LIN {X 0,Y 354.902,Z 376.278,A -85,B 0,C 180,E1 -13615.827,E2 -13615.827} C_VEL
LIN {X 0,Y 354.82,Z 376.288,A -85,B 0,C 180,E1 -13619.682,E2 -13619.682} C_VEL
LIN {X 0,Y 354.808,Z 376.29,A -85,B 0,C 180,E1 -13623.702,E2 -13623.702} C_VEL
LIN {X 0,Y 354.803,Z 376.287,A -85,B 0,C 180,E1 -13626.459,E2 -13626.459} C_VEL
LIN {X 0,Y 354.826,Z 376.289,A -85,B 0,C 180,E1 -13629.423,E2 -13629.423} C_VEL
LIN {X 0,Y 354.79,Z 376.29,A -85,B 0,C 180,E1 -13632.867,E2 -13632.867} C_VEL
LIN {X 0,Y 354.769,Z 376.291,A -85,B 0,C 180,E1 -13636.104,E2 -13636.104} C_VEL
LIN {X 0,Y 354.79,Z 376.293,A -85,B 0,C 180,E1 -13639.179,E2 -13639.179} C_VEL
LIN {X 0,Y 354.809,Z 376.286,A -85,B 0,C 180,E1 -13642.402,E2 -13642.402} C_VEL
LIN {X 0,Y 354.8,Z 376.288,A -85,B 0,C 180,E1 -13643.688,E2 -13643.688} C_VEL
LIN {X 0,Y 354.142,Z 376.373,A -85,B 0,C 180,E1 -13644.636,E2 -13644.636} C_VEL
LIN {X 0,Y 351.287,Z 376.725,A -85,B 0,C 180,E1 -13646.177,E2 -13646.177} C_VEL
LIN {X 0,Y 348.861,Z 377.029,A -85,B 0,C 180,E1 -13647.425,E2 -13647.425} C_VEL
LIN {X 0,Y 347.817,Z 377.158,A -85,B 0,C 180,E1 -13648.39,E2 -13648.39} C_VEL
LIN {X 0,Y 347.732,Z 377.165,A -85,B 0,C 180,E1 -13648.717,E2 -13648.717} C_VEL
LIN {X 0,Y 347.807,Z 377.163,A -85,B 0,C 180,E1 -13650.99,E2 -13650.99} C_VEL
LIN {X 0,Y 347.834,Z 377.155,A -85,B 0,C 180,E1 -13653.608,E2 -13653.608} C_VEL
LIN {X 0,Y 347.791,Z 377.16,A -85,B 0,C 180,E1 -13656.162,E2 -13656.162} C_VEL
LIN {X 0,Y 347.815,Z 377.157,A -85,B 0,C 180,E1 -13659.909,E2 -13659.909} C_VEL
LIN {X 0,Y 347.868,Z 377.152,A -85,B 0,C 180,E1 -13662.359,E2 -13662.359} C_VEL
LIN {X 0,Y 347.899,Z 377.147,A -85,B 0,C 180,E1 -13665.971,E2 -13665.971} C_VEL
LIN {X 0,Y 347.935,Z 377.142,A -85,B 0,C 180,E1 -13669.526,E2 -13669.526} C_VEL
LIN {X 0,Y 348.077,Z 377.125,A -85,B 0,C 180,E1 -13671.875,E2 -13671.875} C_VEL
LIN {X 0,Y 348.07,Z 377.128,A -85,B 0,C 180,E1 -13674.206,E2 -13674.206} C_VEL
LIN {X 0,Y 348.208,Z 377.108,A -85,B 0,C 180,E1 -13677.686,E2 -13677.686} C_VEL
LIN {X 0,Y 348.349,Z 377.092,A -85,B 0,C 180,E1 -13680,E2 -13680} C_VEL
LIN {X 0,Y 348.21,Z 377.112,A -85,B 0,C 180,E1 -13682.313,E2 -13682.313} C_VEL
LIN {X 0,Y 348.108,Z 377.121,A -85,B 0,C 180,E1 -13686.958,E2 -13686.958} C_VEL
LIN {X 0,Y 347.969,Z 377.138,A -85,B 0,C 180,E1 -13689.298,E2 -13689.298} C_VEL
LIN {X 0,Y 347.892,Z 377.149,A -85,B 0,C 180,E1 -13692.839,E2 -13692.839} C_VEL
LIN {X 0,Y 347.841,Z 377.157,A -85,B 0,C 180,E1 -13696.431,E2 -13696.431} C_VEL
LIN {X 0,Y 347.857,Z 377.152,A -85,B 0,C 180,E1 -13698.86,E2 -13698.86} C_VEL
LIN {X 0,Y 347.776,Z 377.164,A -85,B 0,C 180,E1 -13702.579,E2 -13702.579} C_VEL
LIN {X 0,Y 347.814,Z 377.157,A -85,B 0,C 180,E1 -13705.108,E2 -13705.108} C_VEL
LIN {X 0,Y 347.809,Z 377.16,A -85,B 0,C 180,E1 -13707.694,E2 -13707.694} C_VEL
LIN {X 0,Y 347.75,Z 377.168,A -85,B 0,C 180,E1 -13710.348,E2 -13710.348} C_VEL
LIN {X 0,Y 347.749,Z 377.17,A -85,B 0,C 180,E1 -13714.044,E2 -13714.044} C_VEL
LIN {X 0,Y 347.764,Z 377.165,A -85,B 0,C 180,E1 -13717.321,E2 -13717.321} C_VEL
LIN {X 0,Y 347.745,Z 377.167,A -85,B 0,C 180,E1 -13720.295,E2 -13720.295} C_VEL
LIN {X 0,Y 347.726,Z 377.171,A -85,B 0,C 180,E1 -13723.408,E2 -13723.408} C_VEL
LIN {X 0,Y 347.747,Z 377.166,A -85,B 0,C 180,E1 -13726.683,E2 -13726.683} C_VEL
LIN {X 0,Y 347.749,Z 377.166,A -85,B 0,C 180,E1 -13730.173,E2 -13730.173} C_VEL
LIN {X 0,Y 347.822,Z 377.188,A -85,B 0,C 180,E1 -13731.43,E2 -13731.43} C_VEL
LIN {X 0,Y 350.046,Z 388.259,A -85,B 0,C 180,E1 -13735.404,E2 -13735.404} C_VEL
LIN {X 0,Y 352.34,Z 398.991,A -85,B 0,C 180,E1 -13739.06,E2 -13739.06} C_VEL
LIN {X 0,Y 352.6,Z 402.242,A -85,B 0,C 180,E1 -13740.112,E2 -13740.112} C_VEL
LIN {X 0,Y 350.956,Z 413.413,A -85,B 0,C 180,E1 -13743.541,E2 -13743.541} C_VEL
LIN {X 0,Y 349.245,Z 426.523,A -85,B 0,C 180,E1 -13747.521,E2 -13747.521} C_VEL
LIN {X 0,Y 347.88,Z 441.264,A -85,B 0,C 180,E1 -13751.933,E2 -13751.933} C_VEL
LIN {X 0,Y 348.663,Z 454.689,A -85,B 0,C 180,E1 -13752.458,E2 -13752.458} C_VEL
LIN {X 0,Y 349.685,Z 467.492,A -85,B 0,C 180,E1 -13753.207,E2 -13753.207} C_VEL
LIN {X 0,Y 349.831,Z 473.774,A -85,B 0,C 180,E1 -13753.665,E2 -13753.665} C_VEL
LIN {X 0,Y 349.134,Z 485.339,A -85,B 0,C 180,E1 -13754.68,E2 -13754.68} C_VEL
LIN {X 0,Y 348.486,Z 495.132,A -85,B 0,C 180,E1 -13755.772,E2 -13755.772} C_VEL
LIN {X 0,Y 347.817,Z 505.176,A -85,B 0,C 180,E1 -13757.158,E2 -13757.158} C_VEL
LIN {X 0,Y 347.265,Z 513.742,A -85,B 0,C 180,E1 -13758.62,E2 -13758.62} C_VEL
LIN {X 0,Y 346.833,Z 521.96,A -85,B 0,C 180,E1 -13760.377,E2 -13760.377} C_VEL
LIN {X 0,Y 346.716,Z 527.501,A -85,B 0,C 180,E1 -13761.843,E2 -13761.843} C_VEL
LIN {X 0,Y 346.711,Z 533.244,A -85,B 0,C 180,E1 -13763.761,E2 -13763.761} C_VEL
LIN {X 0,Y 346.663,Z 537.853,A -85,B 0,C 180,E1 -13765.931,E2 -13765.931} C_VEL
LIN {X 0,Y 346.843,Z 540.335,A -85,B 0,C 180,E1 -13767.678,E2 -13767.678} C_VEL
LIN {X 0,Y 346.742,Z 541.379,A -85,B 0,C 180,E1 -13768.839,E2 -13768.839} C_VEL
LIN {X 0,Y 346.701,Z 541.955,A -85,B 0,C 180,E1 -13770,E2 -13770} C_VEL
LIN {X 0,Y 346.736,Z 542.121,A -85,B 0,C 180,E1 -13771.162,E2 -13771.162} C_VEL
LIN {X 0,Y 346.686,Z 541.835,A -85,B 0,C 180,E1 -13772.324,E2 -13772.324} C_VEL
LIN {X 0,Y 346.563,Z 541.081,A -85,B 0,C 180,E1 -13773.488,E2 -13773.488} C_VEL
LIN {X 0,Y 346.457,Z 539.915,A -85,B 0,C 180,E1 -13774.654,E2 -13774.654} C_VEL
LIN {X 0,Y 346.429,Z 537.606,A -85,B 0,C 180,E1 -13776.245,E2 -13776.245} C_VEL
LIN {X 0,Y 346.542,Z 533.716,A -85,B 0,C 180,E1 -13778.162,E2 -13778.162} C_VEL
LIN {X 0,Y 346.818,Z 528.987,A -85,B 0,C 180,E1 -13779.919,E2 -13779.919} C_VEL
LIN {X 0,Y 347.561,Z 521.864,A -85,B 0,C 180,E1 -13781.962,E2 -13781.962} C_VEL
LIN {X 0,Y 348.465,Z 514.211,A -85,B 0,C 180,E1 -13783.708,E2 -13783.708} C_VEL
LIN {X 0,Y 349.759,Z 504.664,A -85,B 0,C 180,E1 -13785.441,E2 -13785.441} C_VEL
LIN {X 0,Y 351.134,Z 494.905,A -85,B 0,C 180,E1 -13786.871,E2 -13786.871} C_VEL
LIN {X 0,Y 352.7,Z 484.013,A -85,B 0,C 180,E1 -13788.141,E2 -13788.141} C_VEL
LIN {X 0,Y 353.621,Z 475.22,A -85,B 0,C 180,E1 -13788.993,E2 -13788.993} C_VEL
LIN {X 0,Y 353.744,Z 463.645,A -85,B 0,C 180,E1 -13789.977,E2 -13789.977} C_VEL
LIN {X 0,Y 352.874,Z 453.505,A -85,B 0,C 180,E1 -13790.738,E2 -13790.738} C_VEL
LIN {X 0,Y 350.583,Z 441.519,A -85,B 0,C 180,E1 -13791.563,E2 -13791.563} C_VEL
LIN {X 0,Y 350.029,Z 438.72,A -85,B 0,C 180,E1 -13791.766,E2 -13791.766} C_VEL
LIN {X 0,Y 351.953,Z 427.823,A -85,B 0,C 180,E1 -13795.425,E2 -13795.425} C_VEL
LIN {X 0,Y 354.377,Z 418.278,A -85,B 0,C 180,E1 -13798.889,E2 -13798.889} C_VEL
LIN {X 0,Y 355.825,Z 413.221,A -85,B 0,C 180,E1 -13800.9,E2 -13800.9} C_VEL
LIN {X 0,Y 355.475,Z 409.158,A -85,B 0,C 180,E1 -13802.936,E2 -13802.936} C_VEL
LIN {X 0,Y 354.586,Z 404.655,A -85,B 0,C 180,E1 -13805.646,E2 -13805.646} C_VEL
LIN {X 0,Y 353.52,Z 400.178,A -85,B 0,C 180,E1 -13809.165,E2 -13809.165} C_VEL
LIN {X 0,Y 353.123,Z 398.346,A -85,B 0,C 180,E1 -13811.055,E2 -13811.055} C_VEL
LIN {X 0,Y 352.547,Z 396.189,A -85,B 0,C 180,E1 -13814.245,E2 -13814.245} C_VEL
LIN {X 0,Y 352.194,Z 395.182,A -85,B 0,C 180,E1 -13817.276,E2 -13817.276} C_VEL
LIN {X 0,Y 352.011,Z 395.113,A -85,B 0,C 180,E1 -13820.291,E2 -13820.291} C_VEL
LIN {X 0,Y 351.962,Z 395.849,A -85,B 0,C 180,E1 -13823.199,E2 -13823.199} C_VEL
LIN {X 0,Y 352,Z 397.199,A -85,B 0,C 180,E1 -13826.01,E2 -13826.01} C_VEL
LIN {X 0,Y 352.025,Z 398.061,A -85,B 0,C 180,E1 -13827.382,E2 -13827.382} C_VEL
LIN {X 0,Y 351.653,Z 400.251,A -85,B 0,C 180,E1 -13830.024,E2 -13830.024} C_VEL
LIN {X 0,Y 350.985,Z 402.815,A -85,B 0,C 180,E1 -13832.578,E2 -13832.578} C_VEL
LIN {X 0,Y 350.363,Z 405.632,A -85,B 0,C 180,E1 -13835.087,E2 -13835.087} C_VEL
LIN {X 0,Y 349.584,Z 410.186,A -85,B 0,C 180,E1 -13838.785,E2 -13838.785} C_VEL
LIN {X 0,Y 349.203,Z 413.406,A -85,B 0,C 180,E1 -13841.215,E2 -13841.215} C_VEL
LIN {X 0,Y 348.751,Z 417.005,A -85,B 0,C 180,E1 -13843.681,E2 -13843.681} C_VEL
LIN {X 0,Y 352.118,Z 427.833,A -85,B 0,C 180,E1 -13844.961,E2 -13844.961} C_VEL
LIN {X 0,Y 354.054,Z 437.746,A -85,B 0,C 180,E1 -13846.22,E2 -13846.22} C_VEL
LIN {X 0,Y 354.262,Z 441.119,A -85,B 0,C 180,E1 -13846.667,E2 -13846.667} C_VEL
LIN {X 0,Y 353.026,Z 449.888,A -85,B 0,C 180,E1 -13847.848,E2 -13847.848} C_VEL
LIN {X 0,Y 351.861,Z 457.162,A -85,B 0,C 180,E1 -13849.062,E2 -13849.062} C_VEL
LIN {X 0,Y 350.663,Z 463.864,A -85,B 0,C 180,E1 -13850.483,E2 -13850.483} C_VEL
LIN {X 0,Y 349.641,Z 469.036,A -85,B 0,C 180,E1 -13851.911,E2 -13851.911} C_VEL
LIN {X 0,Y 348.699,Z 473.576,A -85,B 0,C 180,E1 -13853.636,E2 -13853.636} C_VEL
LIN {X 0,Y 347.795,Z 476.569,A -85,B 0,C 180,E1 -13855.364,E2 -13855.364} C_VEL
LIN {X 0,Y 347.324,Z 477.722,A -85,B 0,C 180,E1 -13856.52,E2 -13856.52} C_VEL
LIN {X 0,Y 347.007,Z 478.218,A -85,B 0,C 180,E1 -13857.679,E2 -13857.679} C_VEL
LIN {X 0,Y 346.831,Z 478.063,A -85,B 0,C 180,E1 -13858.839,E2 -13858.839} C_VEL
LIN {X 0,Y 346.758,Z 477.255,A -85,B 0,C 180,E1 -13860,E2 -13860} C_VEL
LIN {X 0,Y 346.746,Z 474.808,A -85,B 0,C 180,E1 -13861.742,E2 -13861.742} C_VEL
LIN {X 0,Y 346.926,Z 470.763,A -85,B 0,C 180,E1 -13863.484,E2 -13863.484} C_VEL
LIN {X 0,Y 347.224,Z 466.034,A -85,B 0,C 180,E1 -13864.935,E2 -13864.935} C_VEL
LIN {X 0,Y 347.466,Z 459.863,A -85,B 0,C 180,E1 -13866.387,E2 -13866.387} C_VEL
LIN {X 0,Y 347.733,Z 452.232,A -85,B 0,C 180,E1 -13867.787,E2 -13867.787} C_VEL
LIN {X 0,Y 348.068,Z 443.808,A -85,B 0,C 180,E1 -13869.003,E2 -13869.003} C_VEL
LIN {X 0,Y 348.565,Z 433.457,A -85,B 0,C 180,E1 -13870.162,E2 -13870.162} C_VEL
LIN {X 0,Y 348.629,Z 426.981,A -85,B 0,C 180,E1 -13870.747,E2 -13870.747} C_VEL
LIN {X 0,Y 347.297,Z 416.48,A -85,B 0,C 180,E1 -13871.527,E2 -13871.527} C_VEL
LIN {X 0,Y 346.726,Z 411.274,A -85,B 0,C 180,E1 -13871.843,E2 -13871.843} C_VEL
LIN {X 0,Y 346.893,Z 405.068,A -85,B 0,C 180,E1 -13875.271,E2 -13875.271} C_VEL
LIN {X 0,Y 347.067,Z 400.434,A -85,B 0,C 180,E1 -13877.873,E2 -13877.873} C_VEL
LIN {X 0,Y 347.299,Z 394.216,A -85,B 0,C 180,E1 -13881.429,E2 -13881.429} C_VEL
LIN {X 0,Y 347.606,Z 387.863,A -85,B 0,C 180,E1 -13885.125,E2 -13885.125} C_VEL
LIN {X 0,Y 348.002,Z 381.36,A -85,B 0,C 180,E1 -13888.992,E2 -13888.992} C_VEL
LIN {X 0,Y 348.044,Z 378.068,A -85,B 0,C 180,E1 -13890.992,E2 -13890.992} C_VEL
LIN {X 0,Y 347.955,Z 377.142,A -85,B 0,C 180,E1 -13891.678,E2 -13891.678} C_VEL
LIN {X 0,Y 347.774,Z 377.162,A -85,B 0,C 180,E1 -13896.065,E2 -13896.065} C_VEL
LIN {X 0,Y 347.755,Z 377.169,A -85,B 0,C 180,E1 -13898.793,E2 -13898.793} C_VEL
LIN {X 0,Y 347.753,Z 377.165,A -85,B 0,C 180,E1 -13901.83,E2 -13901.83} C_VEL
LIN {X 0,Y 347.769,Z 377.166,A -85,B 0,C 180,E1 -13905.017,E2 -13905.017} C_VEL
LIN {X 0,Y 347.753,Z 377.168,A -85,B 0,C 180,E1 -13908.397,E2 -13908.397} C_VEL
LIN {X 0,Y 347.776,Z 377.163,A -85,B 0,C 180,E1 -13912.011,E2 -13912.011} C_VEL
LIN {X 0,Y 347.747,Z 377.165,A -85,B 0,C 180,E1 -13915.536,E2 -13915.536} C_VEL
LIN {X 0,Y 347.748,Z 377.169,A -85,B 0,C 180,E1 -13918.3,E2 -13918.3} C_VEL
LIN {X 0,Y 347.781,Z 377.163,A -85,B 0,C 180,E1 -13920.988,E2 -13920.988} C_VEL
LIN {X 0,Y 347.834,Z 377.155,A -85,B 0,C 180,E1 -13923.608,E2 -13923.608} C_VEL
LIN {X 0,Y 347.792,Z 377.163,A -85,B 0,C 180,E1 -13926.162,E2 -13926.162} C_VEL
LIN {X 0,Y 347.821,Z 377.158,A -85,B 0,C 180,E1 -13929.91,E2 -13929.91} C_VEL
LIN {X 0,Y 347.87,Z 377.155,A -85,B 0,C 180,E1 -13932.359,E2 -13932.359} C_VEL
LIN {X 0,Y 347.9,Z 377.15,A -85,B 0,C 180,E1 -13935.971,E2 -13935.971} C_VEL
LIN {X 0,Y 347.932,Z 377.143,A -85,B 0,C 180,E1 -13939.526,E2 -13939.526} C_VEL
LIN {X 0,Y 348.094,Z 377.122,A -85,B 0,C 180,E1 -13943.042,E2 -13943.042} C_VEL
LIN {X 0,Y 348.21,Z 377.11,A -85,B 0,C 180,E1 -13947.686,E2 -13947.686} C_VEL
LIN {X 0,Y 348.348,Z 377.096,A -85,B 0,C 180,E1 -13950,E2 -13950} C_VEL
LIN {X 0,Y 348.212,Z 377.11,A -85,B 0,C 180,E1 -13952.313,E2 -13952.313} C_VEL
LIN {X 0,Y 348.095,Z 377.122,A -85,B 0,C 180,E1 -13956.958,E2 -13956.958} C_VEL
LIN {X 0,Y 347.933,Z 377.143,A -85,B 0,C 180,E1 -13960.474,E2 -13960.474} C_VEL
LIN {X 0,Y 347.901,Z 377.149,A -85,B 0,C 180,E1 -13964.15,E2 -13964.15} C_VEL
LIN {X 0,Y 347.895,Z 377.148,A -85,B 0,C 180,E1 -13968.291,E2 -13968.291} C_VEL
LIN {X 0,Y 347.8,Z 377.164,A -85,B 0,C 180,E1 -13971.639,E2 -13971.639} C_VEL
LIN {X 0,Y 347.815,Z 377.159,A -85,B 0,C 180,E1 -13975.108,E2 -13975.108} C_VEL
LIN {X 0,Y 347.811,Z 377.162,A -85,B 0,C 180,E1 -13977.694,E2 -13977.694} C_VEL
LIN {X 0,Y 347.751,Z 377.165,A -85,B 0,C 180,E1 -13980.348,E2 -13980.348} C_VEL
LIN {X 0,Y 347.75,Z 377.166,A -85,B 0,C 180,E1 -13984.044,E2 -13984.044} C_VEL
LIN {X 0,Y 347.767,Z 377.168,A -85,B 0,C 180,E1 -13987.32,E2 -13987.32} C_VEL
LIN {X 0,Y 347.735,Z 377.167,A -85,B 0,C 180,E1 -13990.297,E2 -13990.297} C_VEL
LIN {X 0,Y 347.725,Z 377.173,A -85,B 0,C 180,E1 -13993.408,E2 -13993.408} C_VEL
LIN {X 0,Y 347.727,Z 377.169,A -85,B 0,C 180,E1 -13996.686,E2 -13996.686} C_VEL
LIN {X 0,Y 347.749,Z 377.165,A -85,B 0,C 180,E1 -14000.173,E2 -14000.173} C_VEL
LIN {X 0,Y 347.758,Z 377.163,A -85,B 0,C 180,E1 -14003.697,E2 -14003.697} C_VEL
LIN {X 0,Y 347.735,Z 377.172,A -85,B 0,C 180,E1 -14006.928,E2 -14006.928} C_VEL
LIN {X 0,Y 347.732,Z 377.165,A -85,B 0,C 180,E1 -14008.717,E2 -14008.717} C_VEL
LIN {X 0,Y 347.071,Z 377.251,A -85,B 0,C 180,E1 -14009.684,E2 -14009.684} C_VEL
LIN {X 0,Y 344.253,Z 377.604,A -85,B 0,C 180,E1 -14011.259,E2 -14011.259} C_VEL
LIN {X 0,Y 341.868,Z 377.9,A -85,B 0,C 180,E1 -14012.533,E2 -14012.533} C_VEL
LIN {X 0,Y 340.847,Z 378.026,A -85,B 0,C 180,E1 -14013.519,E2 -14013.519} C_VEL
LIN {X 0,Y 340.766,Z 378.035,A -85,B 0,C 180,E1 -14013.852,E2 -14013.852} C_VEL
LIN {X 0,Y 340.731,Z 378.044,A -85,B 0,C 180,E1 -14016.927,E2 -14016.927} C_VEL
LIN {X 0,Y 340.793,Z 378.037,A -85,B 0,C 180,E1 -14020.733,E2 -14020.733} C_VEL
LIN {X 0,Y 340.789,Z 378.034,A -85,B 0,C 180,E1 -14023.219,E2 -14023.219} C_VEL
LIN {X 0,Y 340.849,Z 378.029,A -85,B 0,C 180,E1 -14026.89,E2 -14026.89} C_VEL
LIN {X 0,Y 340.932,Z 378.019,A -85,B 0,C 180,E1 -14030.508,E2 -14030.508} C_VEL
LIN {X 0,Y 341.078,Z 377.999,A -85,B 0,C 180,E1 -14032.898,E2 -14032.898} C_VEL
LIN {X 0,Y 341.17,Z 377.985,A -85,B 0,C 180,E1 -14037.639,E2 -14037.639} C_VEL
LIN {X 0,Y 341.299,Z 377.97,A -85,B 0,C 180,E1 -14040,E2 -14040} C_VEL
LIN {X 0,Y 341.172,Z 377.989,A -85,B 0,C 180,E1 -14042.361,E2 -14042.361} C_VEL
LIN {X 0,Y 341.078,Z 377.996,A -85,B 0,C 180,E1 -14047.102,E2 -14047.102} C_VEL
LIN {X 0,Y 340.873,Z 378.024,A -85,B 0,C 180,E1 -14050.694,E2 -14050.694} C_VEL
LIN {X 0,Y 340.864,Z 378.028,A -85,B 0,C 180,E1 -14054.325,E2 -14054.325} C_VEL
LIN {X 0,Y 340.839,Z 378.029,A -85,B 0,C 180,E1 -14058.467,E2 -14058.467} C_VEL
LIN {X 0,Y 340.755,Z 378.04,A -85,B 0,C 180,E1 -14061.857,E2 -14061.857} C_VEL
LIN {X 0,Y 340.774,Z 378.036,A -85,B 0,C 180,E1 -14065.664,E2 -14065.664} C_VEL
LIN {X 0,Y 340.73,Z 378.042,A -85,B 0,C 180,E1 -14068.321,E2 -14068.321} C_VEL
LIN {X 0,Y 340.699,Z 378.043,A -85,B 0,C 180,E1 -14071.045,E2 -14071.045} C_VEL
LIN {X 0,Y 340.72,Z 378.042,A -85,B 0,C 180,E1 -14075.279,E2 -14075.279} C_VEL
LIN {X 0,Y 340.713,Z 378.043,A -85,B 0,C 180,E1 -14078.386,E2 -14078.386} C_VEL
LIN {X 0,Y 340.704,Z 378.046,A -85,B 0,C 180,E1 -14082.046,E2 -14082.046} C_VEL
LIN {X 0,Y 340.692,Z 378.047,A -85,B 0,C 180,E1 -14085.463,E2 -14085.463} C_VEL
LIN {X 0,Y 340.687,Z 378.044,A -85,B 0,C 180,E1 -14088.691,E2 -14088.691} C_VEL
LIN {X 0,Y 340.785,Z 378.225,A -85,B 0,C 180,E1 -14091.145,E2 -14091.145} C_VEL
LIN {X 0,Y 342.917,Z 388.841,A -85,B 0,C 180,E1 -14095.064,E2 -14095.064} C_VEL
LIN {X 0,Y 345.178,Z 399.465,A -85,B 0,C 180,E1 -14098.776,E2 -14098.776} C_VEL
LIN {X 0,Y 345.588,Z 402.453,A -85,B 0,C 180,E1 -14099.78,E2 -14099.78} C_VEL
LIN {X 0,Y 344.453,Z 410.564,A -85,B 0,C 180,E1 -14102.343,E2 -14102.343} C_VEL
LIN {X 0,Y 342.596,Z 423.628,A -85,B 0,C 180,E1 -14106.42,E2 -14106.42} C_VEL
LIN {X 0,Y 340.988,Z 439.087,A -85,B 0,C 180,E1 -14111.204,E2 -14111.204} C_VEL
LIN {X 0,Y 340.838,Z 440.85,A -85,B 0,C 180,E1 -14111.746,E2 -14111.746} C_VEL
LIN {X 0,Y 341.61,Z 454.921,A -85,B 0,C 180,E1 -14112.335,E2 -14112.335} C_VEL
LIN {X 0,Y 342.593,Z 467.205,A -85,B 0,C 180,E1 -14113.08,E2 -14113.08} C_VEL
LIN {X 0,Y 342.736,Z 474.426,A -85,B 0,C 180,E1 -14113.623,E2 -14113.623} C_VEL
LIN {X 0,Y 342.016,Z 486.398,A -85,B 0,C 180,E1 -14114.738,E2 -14114.738} C_VEL
LIN {X 0,Y 341.208,Z 496.998,A -85,B 0,C 180,E1 -14115.994,E2 -14115.994} C_VEL
LIN {X 0,Y 340.698,Z 505.192,A -85,B 0,C 180,E1 -14117.188,E2 -14117.188} C_VEL
LIN {X 0,Y 340.165,Z 513.608,A -85,B 0,C 180,E1 -14118.681,E2 -14118.681} C_VEL
LIN {X 0,Y 339.77,Z 521.736,A -85,B 0,C 180,E1 -14120.475,E2 -14120.475} C_VEL
LIN {X 0,Y 339.635,Z 528.164,A -85,B 0,C 180,E1 -14122.27,E2 -14122.27} C_VEL
LIN {X 0,Y 339.631,Z 533.126,A -85,B 0,C 180,E1 -14124.061,E2 -14124.061} C_VEL
LIN {X 0,Y 339.612,Z 536.822,A -85,B 0,C 180,E1 -14125.847,E2 -14125.847} C_VEL
LIN {X 0,Y 339.796,Z 539.402,A -85,B 0,C 180,E1 -14127.629,E2 -14127.629} C_VEL
LIN {X 0,Y 339.7,Z 540.52,A -85,B 0,C 180,E1 -14128.815,E2 -14128.815} C_VEL
LIN {X 0,Y 339.656,Z 541.157,A -85,B 0,C 180,E1 -14130,E2 -14130} C_VEL
LIN {X 0,Y 339.69,Z 541.363,A -85,B 0,C 180,E1 -14131.186,E2 -14131.186} C_VEL
LIN {X 0,Y 339.615,Z 541.141,A -85,B 0,C 180,E1 -14132.372,E2 -14132.372} C_VEL
LIN {X 0,Y 339.471,Z 540.445,A -85,B 0,C 180,E1 -14133.561,E2 -14133.561} C_VEL
LIN {X 0,Y 339.383,Z 539.322,A -85,B 0,C 180,E1 -14134.752,E2 -14134.752} C_VEL
LIN {X 0,Y 339.338,Z 537.368,A -85,B 0,C 180,E1 -14136.212,E2 -14136.212} C_VEL
LIN {X 0,Y 339.465,Z 533.307,A -85,B 0,C 180,E1 -14138.333,E2 -14138.333} C_VEL
LIN {X 0,Y 339.762,Z 528.686,A -85,B 0,C 180,E1 -14140.127,E2 -14140.127} C_VEL
LIN {X 0,Y 340.427,Z 522.874,A -85,B 0,C 180,E1 -14141.914,E2 -14141.914} C_VEL
LIN {X 0,Y 341.388,Z 515.604,A -85,B 0,C 180,E1 -14143.695,E2 -14143.695} C_VEL
LIN {X 0,Y 342.654,Z 506.683,A -85,B 0,C 180,E1 -14145.464,E2 -14145.464} C_VEL
LIN {X 0,Y 344.245,Z 496.491,A -85,B 0,C 180,E1 -14147.066,E2 -14147.066} C_VEL
LIN {X 0,Y 345.837,Z 486.287,A -85,B 0,C 180,E1 -14148.36,E2 -14148.36} C_VEL
LIN {X 0,Y 347.039,Z 476.583,A -85,B 0,C 180,E1 -14149.367,E2 -14149.367} C_VEL
LIN {X 0,Y 347.319,Z 464.146,A -85,B 0,C 180,E1 -14150.482,E2 -14150.482} C_VEL
LIN {X 0,Y 346.454,Z 454.046,A -85,B 0,C 180,E1 -14151.295,E2 -14151.295} C_VEL
LIN {X 0,Y 344.138,Z 441.723,A -85,B 0,C 180,E1 -14152.212,E2 -14152.212} C_VEL
LIN {X 0,Y 343.406,Z 438.296,A -85,B 0,C 180,E1 -14152.486,E2 -14152.486} C_VEL
LIN {X 0,Y 345.769,Z 426.618,A -85,B 0,C 180,E1 -14156.577,E2 -14156.577} C_VEL
LIN {X 0,Y 348.525,Z 417.035,A -85,B 0,C 180,E1 -14160.273,E2 -14160.273} C_VEL
LIN {X 0,Y 348.965,Z 415.53,A -85,B 0,C 180,E1 -14160.901,E2 -14160.901} C_VEL
LIN {X 0,Y 348.973,Z 412.801,A -85,B 0,C 180,E1 -14162.238,E2 -14162.238} C_VEL
LIN {X 0,Y 348.102,Z 407.905,A -85,B 0,C 180,E1 -14165.128,E2 -14165.128} C_VEL
LIN {X 0,Y 347.207,Z 404.209,A -85,B 0,C 180,E1 -14167.868,E2 -14167.868} C_VEL
LIN {X 0,Y 346.602,Z 401.436,A -85,B 0,C 180,E1 -14170.456,E2 -14170.456} C_VEL
LIN {X 0,Y 345.992,Z 399.079,A -85,B 0,C 180,E1 -14173.68,E2 -14173.68} C_VEL
LIN {X 0,Y 345.669,Z 397.938,A -85,B 0,C 180,E1 -14176.269,E2 -14176.269} C_VEL
LIN {X 0,Y 345.404,Z 397.514,A -85,B 0,C 180,E1 -14179.375,E2 -14179.375} C_VEL
LIN {X 0,Y 345.281,Z 398.003,A -85,B 0,C 180,E1 -14182.545,E2 -14182.545} C_VEL
LIN {X 0,Y 345.273,Z 399.092,A -85,B 0,C 180,E1 -14185.254,E2 -14185.254} C_VEL
LIN {X 0,Y 345.168,Z 400.776,A -85,B 0,C 180,E1 -14188.036,E2 -14188.036} C_VEL
LIN {X 0,Y 344.654,Z 403.003,A -85,B 0,C 180,E1 -14190.699,E2 -14190.699} C_VEL
LIN {X 0,Y 343.647,Z 406.98,A -85,B 0,C 180,E1 -14194.566,E2 -14194.566} C_VEL
LIN {X 0,Y 342.776,Z 411.44,A -85,B 0,C 180,E1 -14198.343,E2 -14198.343} C_VEL
LIN {X 0,Y 342.075,Z 416.26,A -85,B 0,C 180,E1 -14202.051,E2 -14202.051} C_VEL
LIN {X 0,Y 341.907,Z 417.492,A -85,B 0,C 180,E1 -14202.929,E2 -14202.929} C_VEL
LIN {X 0,Y 345.452,Z 428.369,A -85,B 0,C 180,E1 -14204.296,E2 -14204.296} C_VEL
LIN {X 0,Y 347.205,Z 436.77,A -85,B 0,C 180,E1 -14205.423,E2 -14205.423} C_VEL
LIN {X 0,Y 347.811,Z 442.797,A -85,B 0,C 180,E1 -14206.262,E2 -14206.262} C_VEL
LIN {X 0,Y 346.56,Z 451.024,A -85,B 0,C 180,E1 -14207.408,E2 -14207.408} C_VEL
LIN {X 0,Y 345.091,Z 459.166,A -85,B 0,C 180,E1 -14208.844,E2 -14208.844} C_VEL
LIN {X 0,Y 343.835,Z 465.532,A -85,B 0,C 180,E1 -14210.292,E2 -14210.292} C_VEL
LIN {X 0,Y 342.779,Z 470.521,A -85,B 0,C 180,E1 -14211.748,E2 -14211.748} C_VEL
LIN {X 0,Y 341.762,Z 474.851,A -85,B 0,C 180,E1 -14213.506,E2 -14213.506} C_VEL
LIN {X 0,Y 340.797,Z 477.627,A -85,B 0,C 180,E1 -14215.268,E2 -14215.268} C_VEL
LIN {X 0,Y 340.298,Z 478.646,A -85,B 0,C 180,E1 -14216.448,E2 -14216.448} C_VEL
LIN {X 0,Y 339.966,Z 479.022,A -85,B 0,C 180,E1 -14217.631,E2 -14217.631} C_VEL
LIN {X 0,Y 339.784,Z 478.751,A -85,B 0,C 180,E1 -14218.815,E2 -14218.815} C_VEL
LIN {X 0,Y 339.709,Z 477.828,A -85,B 0,C 180,E1 -14220,E2 -14220} C_VEL
LIN {X 0,Y 339.668,Z 475.203,A -85,B 0,C 180,E1 -14221.779,E2 -14221.779} C_VEL
LIN {X 0,Y 339.844,Z 470.992,A -85,B 0,C 180,E1 -14223.557,E2 -14223.557} C_VEL
LIN {X 0,Y 340.149,Z 466.14,A -85,B 0,C 180,E1 -14225.038,E2 -14225.038} C_VEL
LIN {X 0,Y 340.42,Z 459.811,A -85,B 0,C 180,E1 -14226.52,E2 -14226.52} C_VEL
LIN {X 0,Y 340.662,Z 452.714,A -85,B 0,C 180,E1 -14227.827,E2 -14227.827} C_VEL
LIN {X 0,Y 340.972,Z 444.438,A -85,B 0,C 180,E1 -14229.042,E2 -14229.042} C_VEL
LIN {X 0,Y 341.483,Z 434.114,A -85,B 0,C 180,E1 -14230.225,E2 -14230.225} C_VEL
LIN {X 0,Y 341.588,Z 427.68,A -85,B 0,C 180,E1 -14230.821,E2 -14230.821} C_VEL
LIN {X 0,Y 340.281,Z 417.297,A -85,B 0,C 180,E1 -14231.617,E2 -14231.617} C_VEL
LIN {X 0,Y 339.674,Z 411.564,A -85,B 0,C 180,E1 -14231.979,E2 -14231.979} C_VEL
LIN {X 0,Y 339.842,Z 405.117,A -85,B 0,C 180,E1 -14235.596,E2 -14235.596} C_VEL
LIN {X 0,Y 340.035,Z 399.704,A -85,B 0,C 180,E1 -14238.685,E2 -14238.685} C_VEL
LIN {X 0,Y 340.368,Z 393.216,A -85,B 0,C 180,E1 -14242.457,E2 -14242.457} C_VEL
LIN {X 0,Y 340.666,Z 386.692,A -85,B 0,C 180,E1 -14246.331,E2 -14246.331} C_VEL
LIN {X 0,Y 341.089,Z 380.516,A -85,B 0,C 180,E1 -14250.072,E2 -14250.072} C_VEL
LIN {X 0,Y 340.905,Z 378.02,A -85,B 0,C 180,E1 -14251.716,E2 -14251.716} C_VEL
LIN {X 0,Y 340.724,Z 378.043,A -85,B 0,C 180,E1 -14255.278,E2 -14255.278} C_VEL
LIN {X 0,Y 340.713,Z 378.043,A -85,B 0,C 180,E1 -14258.386,E2 -14258.386} C_VEL
LIN {X 0,Y 340.702,Z 378.043,A -85,B 0,C 180,E1 -14262.046,E2 -14262.046} C_VEL
LIN {X 0,Y 340.686,Z 378.045,A -85,B 0,C 180,E1 -14265.461,E2 -14265.461} C_VEL
LIN {X 0,Y 340.689,Z 378.05,A -85,B 0,C 180,E1 -14268.691,E2 -14268.691} C_VEL
LIN {X 0,Y 340.736,Z 378.039,A -85,B 0,C 180,E1 -14271.773,E2 -14271.773} C_VEL
LIN {X 0,Y 340.726,Z 378.04,A -85,B 0,C 180,E1 -14275.595,E2 -14275.595} C_VEL
LIN {X 0,Y 340.701,Z 378.045,A -85,B 0,C 180,E1 -14278.955,E2 -14278.955} C_VEL
LIN {X 0,Y 340.806,Z 378.031,A -85,B 0,C 180,E1 -14283.02,E2 -14283.02} C_VEL
LIN {X 0,Y 340.759,Z 378.036,A -85,B 0,C 180,E1 -14285.638,E2 -14285.638} C_VEL
LIN {X 0,Y 340.751,Z 378.037,A -85,B 0,C 180,E1 -14289.474,E2 -14289.474} C_VEL
LIN {X 0,Y 340.861,Z 378.026,A -85,B 0,C 180,E1 -14291.984,E2 -14291.984} C_VEL
LIN {X 0,Y 340.872,Z 378.023,A -85,B 0,C 180,E1 -14295.705,E2 -14295.705} C_VEL
LIN {X 0,Y 340.874,Z 378.021,A -85,B 0,C 180,E1 -14299.306,E2 -14299.306} C_VEL
LIN {X 0,Y 341.062,Z 377.998,A -85,B 0,C 180,E1 -14302.898,E2 -14302.898} C_VEL
LIN {X 0,Y 341.171,Z 377.986,A -85,B 0,C 180,E1 -14307.639,E2 -14307.639} C_VEL
LIN {X 0,Y 341.298,Z 377.974,A -85,B 0,C 180,E1 -14310,E2 -14310} C_VEL
LIN {X 0,Y 341.173,Z 377.987,A -85,B 0,C 180,E1 -14312.361,E2 -14312.361} C_VEL
LIN {X 0,Y 341.063,Z 377.998,A -85,B 0,C 180,E1 -14317.102,E2 -14317.102} C_VEL
LIN {X 0,Y 340.875,Z 378.021,A -85,B 0,C 180,E1 -14320.694,E2 -14320.694} C_VEL
LIN {X 0,Y 340.866,Z 378.024,A -85,B 0,C 180,E1 -14324.325,E2 -14324.325} C_VEL
LIN {X 0,Y 340.842,Z 378.026,A -85,B 0,C 180,E1 -14328.467,E2 -14328.467} C_VEL
LIN {X 0,Y 340.756,Z 378.04,A -85,B 0,C 180,E1 -14331.857,E2 -14331.857} C_VEL
LIN {X 0,Y 340.775,Z 378.039,A -85,B 0,C 180,E1 -14335.664,E2 -14335.664} C_VEL
LIN {X 0,Y 340.731,Z 378.04,A -85,B 0,C 180,E1 -14338.321,E2 -14338.321} C_VEL
LIN {X 0,Y 340.7,Z 378.045,A -85,B 0,C 180,E1 -14341.044,E2 -14341.044} C_VEL
LIN {X 0,Y 340.721,Z 378.045,A -85,B 0,C 180,E1 -14345.279,E2 -14345.279} C_VEL
LIN {X 0,Y 340.714,Z 378.041,A -85,B 0,C 180,E1 -14348.386,E2 -14348.386} C_VEL
LIN {X 0,Y 340.701,Z 378.043,A -85,B 0,C 180,E1 -14352.045,E2 -14352.045} C_VEL
LIN {X 0,Y 340.654,Z 378.049,A -85,B 0,C 180,E1 -14356.227,E2 -14356.227} C_VEL
LIN {X 0,Y 340.69,Z 378.045,A -85,B 0,C 180,E1 -14359.753,E2 -14359.753} C_VEL
LIN {X 0,Y 340.707,Z 378.047,A -85,B 0,C 180,E1 -14363.258,E2 -14363.258} C_VEL
LIN {X 0,Y 340.694,Z 378.044,A -85,B 0,C 180,E1 -14366.153,E2 -14366.153} C_VEL
LIN {X 0,Y 340.776,Z 378.034,A -85,B 0,C 180,E1 -14370.332,E2 -14370.332} C_VEL
LIN {X 0,Y 340.766,Z 378.035,A -85,B 0,C 180,E1 -14373.852,E2 -14373.852} C_VEL
LIN {X 0,Y 340.1,Z 378.123,A -85,B 0,C 180,E1 -14374.838,E2 -14374.838} C_VEL
LIN {X 0,Y 337.243,Z 378.482,A -85,B 0,C 180,E1 -14376.441,E2 -14376.441} C_VEL
LIN {X 0,Y 334.817,Z 378.786,A -85,B 0,C 180,E1 -14377.739,E2 -14377.739} C_VEL
LIN {X 0,Y 333.773,Z 378.912,A -85,B 0,C 180,E1 -14378.744,E2 -14378.744} C_VEL
LIN {X 0,Y 333.686,Z 378.92,A -85,B 0,C 180,E1 -14379.084,E2 -14379.084} C_VEL
LIN {X 0,Y 333.795,Z 378.903,A -85,B 0,C 180,E1 -14381.589,E2 -14381.589} C_VEL
LIN {X 0,Y 333.81,Z 378.901,A -85,B 0,C 180,E1 -14385.576,E2 -14385.576} C_VEL
LIN {X 0,Y 333.84,Z 378.9,A -85,B 0,C 180,E1 -14389.078,E2 -14389.078} C_VEL
LIN {X 0,Y 334.028,Z 378.879,A -85,B 0,C 180,E1 -14392.747,E2 -14392.747} C_VEL
LIN {X 0,Y 333.812,Z 378.902,A -85,B 0,C 180,E1 -14395.169,E2 -14395.169} C_VEL
LIN {X 0,Y 334.107,Z 378.864,A -85,B 0,C 180,E1 -14397.589,E2 -14397.589} C_VEL
LIN {X 0,Y 334.25,Z 378.848,A -85,B 0,C 180,E1 -14400,E2 -14400} C_VEL
LIN {X 0,Y 334.133,Z 378.866,A -85,B 0,C 180,E1 -14402.411,E2 -14402.411} C_VEL
LIN {X 0,Y 334.028,Z 378.874,A -85,B 0,C 180,E1 -14407.252,E2 -14407.252} C_VEL
LIN {X 0,Y 333.836,Z 378.899,A -85,B 0,C 180,E1 -14410.922,E2 -14410.922} C_VEL
LIN {X 0,Y 333.81,Z 378.904,A -85,B 0,C 180,E1 -14414.634,E2 -14414.634} C_VEL
LIN {X 0,Y 333.798,Z 378.904,A -85,B 0,C 180,E1 -14418.655,E2 -14418.655} C_VEL
LIN {X 0,Y 333.694,Z 378.92,A -85,B 0,C 180,E1 -14422.278,E2 -14422.278} C_VEL
LIN {X 0,Y 333.736,Z 378.914,A -85,B 0,C 180,E1 -14426.246,E2 -14426.246} C_VEL
LIN {X 0,Y 333.691,Z 378.916,A -85,B 0,C 180,E1 -14428.974,E2 -14428.974} C_VEL
LIN {X 0,Y 333.647,Z 378.922,A -85,B 0,C 180,E1 -14432.588,E2 -14432.588} C_VEL
LIN {X 0,Y 333.678,Z 378.921,A -85,B 0,C 180,E1 -14436.139,E2 -14436.139} C_VEL
LIN {X 0,Y 333.651,Z 378.922,A -85,B 0,C 180,E1 -14439.192,E2 -14439.192} C_VEL
LIN {X 0,Y 333.637,Z 378.923,A -85,B 0,C 180,E1 -14442.501,E2 -14442.501} C_VEL
LIN {X 0,Y 333.636,Z 378.927,A -85,B 0,C 180,E1 -14445.962,E2 -14445.962} C_VEL
LIN {X 0,Y 333.648,Z 378.924,A -85,B 0,C 180,E1 -14449.315,E2 -14449.315} C_VEL
LIN {X 0,Y 333.702,Z 378.994,A -85,B 0,C 180,E1 -14450.767,E2 -14450.767} C_VEL
LIN {X 0,Y 335.438,Z 387.728,A -85,B 0,C 180,E1 -14454.081,E2 -14454.081} C_VEL
LIN {X 0,Y 337.223,Z 396.276,A -85,B 0,C 180,E1 -14457.19,E2 -14457.19} C_VEL
LIN {X 0,Y 338.556,Z 402.642,A -85,B 0,C 180,E1 -14459.43,E2 -14459.43} C_VEL
LIN {X 0,Y 338.164,Z 406.782,A -85,B 0,C 180,E1 -14460.795,E2 -14460.795} C_VEL
LIN {X 0,Y 335.993,Z 420.715,A -85,B 0,C 180,E1 -14465.27,E2 -14465.27} C_VEL
LIN {X 0,Y 334.282,Z 434.638,A -85,B 0,C 180,E1 -14469.702,E2 -14469.702} C_VEL
LIN {X 0,Y 333.759,Z 440.578,A -85,B 0,C 180,E1 -14471.587,E2 -14471.587} C_VEL
LIN {X 0,Y 334.52,Z 454.511,A -85,B 0,C 180,E1 -14472.185,E2 -14472.185} C_VEL
LIN {X 0,Y 335.437,Z 466.721,A -85,B 0,C 180,E1 -14472.943,E2 -14472.943} C_VEL
LIN {X 0,Y 335.631,Z 474.901,A -85,B 0,C 180,E1 -14473.579,E2 -14473.579} C_VEL
LIN {X 0,Y 334.914,Z 486.441,A -85,B 0,C 180,E1 -14474.7,E2 -14474.7} C_VEL
LIN {X 0,Y 334.118,Z 497.066,A -85,B 0,C 180,E1 -14476.002,E2 -14476.002} C_VEL
LIN {X 0,Y 333.594,Z 505.134,A -85,B 0,C 180,E1 -14477.22,E2 -14477.22} C_VEL
LIN {X 0,Y 333.08,Z 513.427,A -85,B 0,C 180,E1 -14478.745,E2 -14478.745} C_VEL
LIN {X 0,Y 332.69,Z 521.463,A -85,B 0,C 180,E1 -14480.577,E2 -14480.577} C_VEL
LIN {X 0,Y 332.603,Z 526.842,A -85,B 0,C 180,E1 -14482.106,E2 -14482.106} C_VEL
LIN {X 0,Y 332.582,Z 531.962,A -85,B 0,C 180,E1 -14483.935,E2 -14483.935} C_VEL
LIN {X 0,Y 332.566,Z 535.77,A -85,B 0,C 180,E1 -14485.758,E2 -14485.758} C_VEL
LIN {X 0,Y 332.75,Z 538.452,A -85,B 0,C 180,E1 -14487.579,E2 -14487.579} C_VEL
LIN {X 0,Y 332.658,Z 539.616,A -85,B 0,C 180,E1 -14488.79,E2 -14488.79} C_VEL
LIN {X 0,Y 332.612,Z 540.346,A -85,B 0,C 180,E1 -14490,E2 -14490} C_VEL
LIN {X 0,Y 332.644,Z 540.6,A -85,B 0,C 180,E1 -14491.211,E2 -14491.211} C_VEL
LIN {X 0,Y 332.544,Z 540.42,A -85,B 0,C 180,E1 -14492.423,E2 -14492.423} C_VEL
LIN {X 0,Y 332.38,Z 539.81,A -85,B 0,C 180,E1 -14493.637,E2 -14493.637} C_VEL
LIN {X 0,Y 332.311,Z 538.738,A -85,B 0,C 180,E1 -14494.853,E2 -14494.853} C_VEL
LIN {X 0,Y 332.257,Z 537.082,A -85,B 0,C 180,E1 -14496.194,E2 -14496.194} C_VEL
LIN {X 0,Y 332.361,Z 534.184,A -85,B 0,C 180,E1 -14497.9,E2 -14497.9} C_VEL
LIN {X 0,Y 332.584,Z 530.057,A -85,B 0,C 180,E1 -14499.733,E2 -14499.733} C_VEL
LIN {X 0,Y 333.28,Z 523.773,A -85,B 0,C 180,E1 -14501.865,E2 -14501.865} C_VEL
LIN {X 0,Y 334.297,Z 516.96,A -85,B 0,C 180,E1 -14503.681,E2 -14503.681} C_VEL
LIN {X 0,Y 335.37,Z 509.826,A -85,B 0,C 180,E1 -14505.241,E2 -14505.241} C_VEL
LIN {X 0,Y 336.746,Z 501.873,A -85,B 0,C 180,E1 -14506.677,E2 -14506.677} C_VEL
LIN {X 0,Y 338.4,Z 491.861,A -85,B 0,C 180,E1 -14508.151,E2 -14508.151} C_VEL
LIN {X 0,Y 340.179,Z 480.799,A -85,B 0,C 180,E1 -14509.46,E2 -14509.46} C_VEL
LIN {X 0,Y 340.965,Z 468.298,A -85,B 0,C 180,E1 -14510.697,E2 -14510.697} C_VEL
LIN {X 0,Y 340.525,Z 458.516,A -85,B 0,C 180,E1 -14511.561,E2 -14511.561} C_VEL
LIN {X 0,Y 338.782,Z 446.86,A -85,B 0,C 180,E1 -14512.525,E2 -14512.525} C_VEL
LIN {X 0,Y 336.794,Z 437.989,A -85,B 0,C 180,E1 -14513.212,E2 -14513.212} C_VEL
LIN {X 0,Y 339.198,Z 427.274,A -85,B 0,C 180,E1 -14517.118,E2 -14517.118} C_VEL
LIN {X 0,Y 342.094,Z 417.862,A -85,B 0,C 180,E1 -14520.904,E2 -14520.904} C_VEL
LIN {X 0,Y 342.161,Z 414.424,A -85,B 0,C 180,E1 -14522.633,E2 -14522.633} C_VEL
LIN {X 0,Y 341.421,Z 410.245,A -85,B 0,C 180,E1 -14525.196,E2 -14525.196} C_VEL
LIN {X 0,Y 340.45,Z 406.182,A -85,B 0,C 180,E1 -14528.331,E2 -14528.331} C_VEL
LIN {X 0,Y 339.806,Z 403.154,A -85,B 0,C 180,E1 -14531.44,E2 -14531.44} C_VEL
LIN {X 0,Y 339.232,Z 401.064,A -85,B 0,C 180,E1 -14534.781,E2 -14534.781} C_VEL
LIN {X 0,Y 339,Z 400.361,A -85,B 0,C 180,E1 -14536.832,E2 -14536.832} C_VEL
LIN {X 0,Y 338.718,Z 400.061,A -85,B 0,C 180,E1 -14540.149,E2 -14540.149} C_VEL
LIN {X 0,Y 338.585,Z 400.549,A -85,B 0,C 180,E1 -14542.99,E2 -14542.99} C_VEL
LIN {X 0,Y 338.554,Z 401.855,A -85,B 0,C 180,E1 -14546.136,E2 -14546.136} C_VEL
LIN {X 0,Y 338.335,Z 403.498,A -85,B 0,C 180,E1 -14548.714,E2 -14548.714} C_VEL
LIN {X 0,Y 337.703,Z 405.773,A -85,B 0,C 180,E1 -14551.402,E2 -14551.402} C_VEL
LIN {X 0,Y 336.968,Z 408.387,A -85,B 0,C 180,E1 -14554.024,E2 -14554.024} C_VEL
LIN {X 0,Y 335.985,Z 412.741,A -85,B 0,C 180,E1 -14557.882,E2 -14557.882} C_VEL
LIN {X 0,Y 335.235,Z 417.466,A -85,B 0,C 180,E1 -14561.671,E2 -14561.671} C_VEL
LIN {X 0,Y 335.18,Z 418.201,A -85,B 0,C 180,E1 -14562.123,E2 -14562.123} C_VEL
LIN {X 0,Y 338.663,Z 428.721,A -85,B 0,C 180,E1 -14563.551,E2 -14563.551} C_VEL
LIN {X 0,Y 340.654,Z 437.221,A -85,B 0,C 180,E1 -14564.75,E2 -14564.75} C_VEL
LIN {X 0,Y 341.401,Z 444.612,A -85,B 0,C 180,E1 -14565.849,E2 -14565.849} C_VEL
LIN {X 0,Y 339.884,Z 453.43,A -85,B 0,C 180,E1 -14567.157,E2 -14567.157} C_VEL
LIN {X 0,Y 338.362,Z 461.22,A -85,B 0,C 180,E1 -14568.62,E2 -14568.62} C_VEL
LIN {X 0,Y 337.048,Z 467.291,A -85,B 0,C 180,E1 -14570.094,E2 -14570.094} C_VEL
LIN {X 0,Y 335.912,Z 471.983,A -85,B 0,C 180,E1 -14571.579,E2 -14571.579} C_VEL
LIN {X 0,Y 334.826,Z 476.073,A -85,B 0,C 180,E1 -14573.371,E2 -14573.371} C_VEL
LIN {X 0,Y 333.797,Z 478.666,A -85,B 0,C 180,E1 -14575.169,E2 -14575.169} C_VEL
LIN {X 0,Y 333.274,Z 479.572,A -85,B 0,C 180,E1 -14576.373,E2 -14576.373} C_VEL
LIN {X 0,Y 332.928,Z 479.829,A -85,B 0,C 180,E1 -14577.58,E2 -14577.58} C_VEL
LIN {X 0,Y 332.738,Z 479.433,A -85,B 0,C 180,E1 -14578.79,E2 -14578.79} C_VEL
LIN {X 0,Y 332.644,Z 478.389,A -85,B 0,C 180,E1 -14580,E2 -14580} C_VEL
LIN {X 0,Y 332.594,Z 475.587,A -85,B 0,C 180,E1 -14581.816,E2 -14581.816} C_VEL
LIN {X 0,Y 332.762,Z 471.186,A -85,B 0,C 180,E1 -14583.633,E2 -14583.633} C_VEL
LIN {X 0,Y 333.076,Z 466.139,A -85,B 0,C 180,E1 -14585.145,E2 -14585.145} C_VEL
LIN {X 0,Y 333.355,Z 459.617,A -85,B 0,C 180,E1 -14586.659,E2 -14586.659} C_VEL
LIN {X 0,Y 333.621,Z 451.88,A -85,B 0,C 180,E1 -14588.069,E2 -14588.069} C_VEL
LIN {X 0,Y 333.948,Z 443.876,A -85,B 0,C 180,E1 -14589.234,E2 -14589.234} C_VEL
LIN {X 0,Y 334.404,Z 434.772,A -85,B 0,C 180,E1 -14590.291,E2 -14590.291} C_VEL
LIN {X 0,Y 334.529,Z 428.377,A -85,B 0,C 180,E1 -14590.899,E2 -14590.899} C_VEL
LIN {X 0,Y 333.251,Z 418.118,A -85,B 0,C 180,E1 -14591.712,E2 -14591.712} C_VEL
LIN {X 0,Y 332.611,Z 411.84,A -85,B 0,C 180,E1 -14592.121,E2 -14592.121} C_VEL
LIN {X 0,Y 332.749,Z 406.227,A -85,B 0,C 180,E1 -14595.308,E2 -14595.308} C_VEL
LIN {X 0,Y 332.947,Z 400.778,A -85,B 0,C 180,E1 -14598.459,E2 -14598.459} C_VEL
LIN {X 0,Y 333.222,Z 394.982,A -85,B 0,C 180,E1 -14601.873,E2 -14601.873} C_VEL
LIN {X 0,Y 333.568,Z 388.771,A -85,B 0,C 180,E1 -14605.589,E2 -14605.589} C_VEL
LIN {X 0,Y 334.003,Z 382.163,A -85,B 0,C 180,E1 -14609.636,E2 -14609.636} C_VEL
LIN {X 0,Y 333.86,Z 378.897,A -85,B 0,C 180,E1 -14611.754,E2 -14611.754} C_VEL
LIN {X 0,Y 333.68,Z 378.918,A -85,B 0,C 180,E1 -14616.139,E2 -14616.139} C_VEL
LIN {X 0,Y 333.649,Z 378.924,A -85,B 0,C 180,E1 -14619.192,E2 -14619.192} C_VEL
LIN {X 0,Y 333.636,Z 378.926,A -85,B 0,C 180,E1 -14622.5,E2 -14622.5} C_VEL
LIN {X 0,Y 333.624,Z 378.925,A -85,B 0,C 180,E1 -14625.959,E2 -14625.959} C_VEL
LIN {X 0,Y 333.65,Z 378.922,A -85,B 0,C 180,E1 -14629.315,E2 -14629.315} C_VEL
LIN {X 0,Y 333.668,Z 378.92,A -85,B 0,C 180,E1 -14633.168,E2 -14633.168} C_VEL
LIN {X 0,Y 333.677,Z 378.918,A -85,B 0,C 180,E1 -14635.341,E2 -14635.341} C_VEL
LIN {X 0,Y 333.693,Z 378.916,A -85,B 0,C 180,E1 -14639.637,E2 -14639.637} C_VEL
LIN {X 0,Y 333.743,Z 378.915,A -85,B 0,C 180,E1 -14642.401,E2 -14642.401} C_VEL
LIN {X 0,Y 333.73,Z 378.912,A -85,B 0,C 180,E1 -14645.091,E2 -14645.091} C_VEL
LIN {X 0,Y 333.685,Z 378.918,A -85,B 0,C 180,E1 -14649.019,E2 -14649.019} C_VEL
LIN {X 0,Y 333.798,Z 378.903,A -85,B 0,C 180,E1 -14651.59,E2 -14651.59} C_VEL
LIN {X 0,Y 333.811,Z 378.902,A -85,B 0,C 180,E1 -14655.577,E2 -14655.577} C_VEL
LIN {X 0,Y 333.837,Z 378.898,A -85,B 0,C 180,E1 -14659.078,E2 -14659.078} C_VEL
LIN {X 0,Y 334.009,Z 378.877,A -85,B 0,C 180,E1 -14662.747,E2 -14662.747} C_VEL
LIN {X 0,Y 333.812,Z 378.901,A -85,B 0,C 180,E1 -14665.169,E2 -14665.169} C_VEL
LIN {X 0,Y 334.109,Z 378.866,A -85,B 0,C 180,E1 -14667.589,E2 -14667.589} C_VEL
LIN {X 0,Y 334.249,Z 378.852,A -85,B 0,C 180,E1 -14670,E2 -14670} C_VEL
LIN {X 0,Y 334.111,Z 378.866,A -85,B 0,C 180,E1 -14672.411,E2 -14672.411} C_VEL
LIN {X 0,Y 334.018,Z 378.88,A -85,B 0,C 180,E1 -14676.039,E2 -14676.039} C_VEL
LIN {X 0,Y 333.988,Z 378.88,A -85,B 0,C 180,E1 -14678.501,E2 -14678.501} C_VEL
LIN {X 0,Y 333.795,Z 378.906,A -85,B 0,C 180,E1 -14682.154,E2 -14682.154} C_VEL
LIN {X 0,Y 333.781,Z 378.909,A -85,B 0,C 180,E1 -14685.886,E2 -14685.886} C_VEL
LIN {X 0,Y 333.801,Z 378.902,A -85,B 0,C 180,E1 -14688.656,E2 -14688.656} C_VEL
LIN {X 0,Y 333.695,Z 378.916,A -85,B 0,C 180,E1 -14692.278,E2 -14692.278} C_VEL
LIN {X 0,Y 333.738,Z 378.911,A -85,B 0,C 180,E1 -14696.246,E2 -14696.246} C_VEL
LIN {X 0,Y 333.692,Z 378.917,A -85,B 0,C 180,E1 -14698.974,E2 -14698.974} C_VEL
LIN {X 0,Y 333.646,Z 378.922,A -85,B 0,C 180,E1 -14702.587,E2 -14702.587} C_VEL
LIN {X 0,Y 333.679,Z 378.918,A -85,B 0,C 180,E1 -14706.139,E2 -14706.139} C_VEL
LIN {X 0,Y 333.649,Z 378.926,A -85,B 0,C 180,E1 -14709.192,E2 -14709.192} C_VEL
LIN {X 0,Y 333.634,Z 378.923,A -85,B 0,C 180,E1 -14712.5,E2 -14712.5} C_VEL
LIN {X 0,Y 333.598,Z 378.928,A -85,B 0,C 180,E1 -14715.955,E2 -14715.955} C_VEL
LIN {X 0,Y 333.649,Z 378.926,A -85,B 0,C 180,E1 -14719.315,E2 -14719.315} C_VEL
LIN {X 0,Y 333.667,Z 378.924,A -85,B 0,C 180,E1 -14723.168,E2 -14723.168} C_VEL
LIN {X 0,Y 333.676,Z 378.921,A -85,B 0,C 180,E1 -14725.341,E2 -14725.341} C_VEL
LIN {X 0,Y 333.704,Z 378.915,A -85,B 0,C 180,E1 -14729.71,E2 -14729.71} C_VEL
LIN {X 0,Y 333.745,Z 378.91,A -85,B 0,C 180,E1 -14732.401,E2 -14732.401} C_VEL
LIN {X 0,Y 333.729,Z 378.915,A -85,B 0,C 180,E1 -14735.091,E2 -14735.091} C_VEL
LIN {X 0,Y 333.686,Z 378.92,A -85,B 0,C 180,E1 -14739.084,E2 -14739.084} C_VEL
LIN {X 0,Y 333.017,Z 379.002,A -85,B 0,C 180,E1 -14740.092,E2 -14740.092} C_VEL
LIN {X 0,Y 330.186,Z 379.353,A -85,B 0,C 180,E1 -14741.734,E2 -14741.734} C_VEL
LIN {X 0,Y 327.802,Z 379.653,A -85,B 0,C 180,E1 -14743.063,E2 -14743.063} C_VEL
LIN {X 0,Y 326.797,Z 379.775,A -85,B 0,C 180,E1 -14744.091,E2 -14744.091} C_VEL
LIN {X 0,Y 326.724,Z 379.783,A -85,B 0,C 180,E1 -14744.44,E2 -14744.44} C_VEL
LIN {X 0,Y 326.741,Z 379.782,A -85,B 0,C 180,E1 -14747.579,E2 -14747.579} C_VEL
LIN {X 0,Y 326.93,Z 379.758,A -85,B 0,C 180,E1 -14751.44,E2 -14751.44} C_VEL
LIN {X 0,Y 326.998,Z 379.75,A -85,B 0,C 180,E1 -14753.831,E2 -14753.831} C_VEL
LIN {X 0,Y 327.048,Z 379.743,A -85,B 0,C 180,E1 -14757.537,E2 -14757.537} C_VEL
LIN {X 0,Y 327.201,Z 379.726,A -85,B 0,C 180,E1 -14760,E2 -14760} C_VEL
LIN {X 0,Y 327.07,Z 379.746,A -85,B 0,C 180,E1 -14762.463,E2 -14762.463} C_VEL
LIN {X 0,Y 326.998,Z 379.753,A -85,B 0,C 180,E1 -14766.169,E2 -14766.169} C_VEL
LIN {X 0,Y 326.916,Z 379.763,A -85,B 0,C 180,E1 -14768.655,E2 -14768.655} C_VEL
LIN {X 0,Y 326.737,Z 379.787,A -85,B 0,C 180,E1 -14772.421,E2 -14772.421} C_VEL
LIN {X 0,Y 326.756,Z 379.78,A -85,B 0,C 180,E1 -14774.957,E2 -14774.957} C_VEL
LIN {X 0,Y 326.735,Z 379.783,A -85,B 0,C 180,E1 -14778.838,E2 -14778.838} C_VEL
LIN {X 0,Y 326.622,Z 379.797,A -85,B 0,C 180,E1 -14782.787,E2 -14782.787} C_VEL
LIN {X 0,Y 326.691,Z 379.789,A -85,B 0,C 180,E1 -14785.484,E2 -14785.484} C_VEL
LIN {X 0,Y 326.649,Z 379.796,A -85,B 0,C 180,E1 -14789.66,E2 -14789.66} C_VEL
LIN {X 0,Y 326.62,Z 379.797,A -85,B 0,C 180,E1 -14792.947,E2 -14792.947} C_VEL
LIN {X 0,Y 326.614,Z 379.8,A -85,B 0,C 180,E1 -14795.52,E2 -14795.52} C_VEL
LIN {X 0,Y 326.615,Z 379.798,A -85,B 0,C 180,E1 -14799.228,E2 -14799.228} C_VEL
LIN {X 0,Y 326.585,Z 379.801,A -85,B 0,C 180,E1 -14802.973,E2 -14802.973} C_VEL
LIN {X 0,Y 326.596,Z 379.8,A -85,B 0,C 180,E1 -14807.024,E2 -14807.024} C_VEL
LIN {X 0,Y 326.639,Z 379.829,A -85,B 0,C 180,E1 -14810.397,E2 -14810.397} C_VEL
LIN {X 0,Y 328.392,Z 388.607,A -85,B 0,C 180,E1 -14813.823,E2 -14813.823} C_VEL
LIN {X 0,Y 330.254,Z 397.483,A -85,B 0,C 180,E1 -14817.135,E2 -14817.135} C_VEL
LIN {X 0,Y 331.551,Z 403.829,A -85,B 0,C 180,E1 -14819.42,E2 -14819.42} C_VEL
LIN {X 0,Y 330.744,Z 409.852,A -85,B 0,C 180,E1 -14821.438,E2 -14821.438} C_VEL
LIN {X 0,Y 328.844,Z 421.781,A -85,B 0,C 180,E1 -14825.37,E2 -14825.37} C_VEL
LIN {X 0,Y 327.132,Z 435.601,A -85,B 0,C 180,E1 -14829.895,E2 -14829.895} C_VEL
LIN {X 0,Y 326.707,Z 440.499,A -85,B 0,C 180,E1 -14831.46,E2 -14831.46} C_VEL
LIN {X 0,Y 327.354,Z 452.908,A -85,B 0,C 180,E1 -14831.984,E2 -14831.984} C_VEL
LIN {X 0,Y 328.229,Z 464.928,A -85,B 0,C 180,E1 -14832.717,E2 -14832.717} C_VEL
LIN {X 0,Y 328.62,Z 473.359,A -85,B 0,C 180,E1 -14833.379,E2 -14833.379} C_VEL
LIN {X 0,Y 327.933,Z 484.432,A -85,B 0,C 180,E1 -14834.445,E2 -14834.445} C_VEL
LIN {X 0,Y 327.185,Z 494.727,A -85,B 0,C 180,E1 -14835.699,E2 -14835.699} C_VEL
LIN {X 0,Y 326.655,Z 503.085,A -85,B 0,C 180,E1 -14836.944,E2 -14836.944} C_VEL
LIN {X 0,Y 326.09,Z 511.683,A -85,B 0,C 180,E1 -14838.501,E2 -14838.501} C_VEL
LIN {X 0,Y 325.663,Z 519.907,A -85,B 0,C 180,E1 -14840.372,E2 -14840.372} C_VEL
LIN {X 0,Y 325.549,Z 525.442,A -85,B 0,C 180,E1 -14841.934,E2 -14841.934} C_VEL
LIN {X 0,Y 325.538,Z 530.731,A -85,B 0,C 180,E1 -14843.803,E2 -14843.803} C_VEL
LIN {X 0,Y 325.522,Z 534.689,A -85,B 0,C 180,E1 -14845.666,E2 -14845.666} C_VEL
LIN {X 0,Y 325.705,Z 537.484,A -85,B 0,C 180,E1 -14847.527,E2 -14847.527} C_VEL
LIN {X 0,Y 325.617,Z 538.698,A -85,B 0,C 180,E1 -14848.763,E2 -14848.763} C_VEL
LIN {X 0,Y 325.569,Z 539.487,A -85,B 0,C 180,E1 -14850,E2 -14850} C_VEL
LIN {X 0,Y 325.597,Z 539.83,A -85,B 0,C 180,E1 -14851.237,E2 -14851.237} C_VEL
LIN {X 0,Y 325.473,Z 539.694,A -85,B 0,C 180,E1 -14852.475,E2 -14852.475} C_VEL
LIN {X 0,Y 325.294,Z 539.141,A -85,B 0,C 180,E1 -14853.716,E2 -14853.716} C_VEL
LIN {X 0,Y 325.241,Z 538.16,A -85,B 0,C 180,E1 -14854.959,E2 -14854.959} C_VEL
LIN {X 0,Y 325.193,Z 536.723,A -85,B 0,C 180,E1 -14856.204,E2 -14856.204} C_VEL
LIN {X 0,Y 325.265,Z 533.761,A -85,B 0,C 180,E1 -14858.074,E2 -14858.074} C_VEL
LIN {X 0,Y 325.53,Z 529.76,A -85,B 0,C 180,E1 -14859.946,E2 -14859.946} C_VEL
LIN {X 0,Y 326.148,Z 524.637,A -85,B 0,C 180,E1 -14861.813,E2 -14861.813} C_VEL
LIN {X 0,Y 327.204,Z 518.263,A -85,B 0,C 180,E1 -14863.667,E2 -14863.667} C_VEL
LIN {X 0,Y 328.439,Z 510.567,A -85,B 0,C 180,E1 -14865.466,E2 -14865.466} C_VEL
LIN {X 0,Y 329.963,Z 502.366,A -85,B 0,C 180,E1 -14867.03,E2 -14867.03} C_VEL
LIN {X 0,Y 331.718,Z 492.747,A -85,B 0,C 180,E1 -14868.53,E2 -14868.53} C_VEL
LIN {X 0,Y 333.792,Z 480.781,A -85,B 0,C 180,E1 -14870.008,E2 -14870.008} C_VEL
LIN {X 0,Y 334.588,Z 468.37,A -85,B 0,C 180,E1 -14871.299,E2 -14871.299} C_VEL
LIN {X 0,Y 334.268,Z 459.652,A -85,B 0,C 180,E1 -14872.118,E2 -14872.118} C_VEL
LIN {X 0,Y 332.763,Z 448.921,A -85,B 0,C 180,E1 -14873.081,E2 -14873.081} C_VEL
LIN {X 0,Y 330.285,Z 437.507,A -85,B 0,C 180,E1 -14874.065,E2 -14874.065} C_VEL
LIN {X 0,Y 333.121,Z 426.341,A -85,B 0,C 180,E1 -14878.34,E2 -14878.34} C_VEL
LIN {X 0,Y 335.005,Z 420.75,A -85,B 0,C 180,E1 -14880.668,E2 -14880.668} C_VEL
LIN {X 0,Y 335.485,Z 418.752,A -85,B 0,C 180,E1 -14881.582,E2 -14881.582} C_VEL
LIN {X 0,Y 335.337,Z 416.1,A -85,B 0,C 180,E1 -14883.037,E2 -14883.037} C_VEL
LIN {X 0,Y 334.801,Z 412.911,A -85,B 0,C 180,E1 -14885.048,E2 -14885.048} C_VEL
LIN {X 0,Y 333.972,Z 409.564,A -85,B 0,C 180,E1 -14887.609,E2 -14887.609} C_VEL
LIN {X 0,Y 333.292,Z 406.254,A -85,B 0,C 180,E1 -14890.82,E2 -14890.82} C_VEL
LIN {X 0,Y 332.677,Z 403.951,A -85,B 0,C 180,E1 -14894.199,E2 -14894.199} C_VEL
LIN {X 0,Y 332.291,Z 402.791,A -85,B 0,C 180,E1 -14897.405,E2 -14897.405} C_VEL
LIN {X 0,Y 332.036,Z 402.575,A -85,B 0,C 180,E1 -14900.581,E2 -14900.581} C_VEL
LIN {X 0,Y 331.878,Z 403.153,A -85,B 0,C 180,E1 -14903.634,E2 -14903.634} C_VEL
LIN {X 0,Y 331.788,Z 404.416,A -85,B 0,C 180,E1 -14906.582,E2 -14906.582} C_VEL
LIN {X 0,Y 331.663,Z 405.252,A -85,B 0,C 180,E1 -14908.011,E2 -14908.011} C_VEL
LIN {X 0,Y 331.086,Z 407.366,A -85,B 0,C 180,E1 -14910.776,E2 -14910.776} C_VEL
LIN {X 0,Y 330.291,Z 409.868,A -85,B 0,C 180,E1 -14913.459,E2 -14913.459} C_VEL
LIN {X 0,Y 329.23,Z 414.082,A -85,B 0,C 180,E1 -14917.403,E2 -14917.403} C_VEL
LIN {X 0,Y 328.429,Z 418.652,A -85,B 0,C 180,E1 -14921.21,E2 -14921.21} C_VEL
LIN {X 0,Y 332.237,Z 429.951,A -85,B 0,C 180,E1 -14922.858,E2 -14922.858} C_VEL
LIN {X 0,Y 334.404,Z 439.377,A -85,B 0,C 180,E1 -14924.301,E2 -14924.301} C_VEL
LIN {X 0,Y 335.013,Z 446.555,A -85,B 0,C 180,E1 -14925.42,E2 -14925.42} C_VEL
LIN {X 0,Y 333.575,Z 454.222,A -85,B 0,C 180,E1 -14926.6,E2 -14926.6} C_VEL
LIN {X 0,Y 331.93,Z 461.909,A -85,B 0,C 180,E1 -14928.086,E2 -14928.086} C_VEL
LIN {X 0,Y 330.254,Z 469.017,A -85,B 0,C 180,E1 -14929.889,E2 -14929.889} C_VEL
LIN {X 0,Y 329.06,Z 473.501,A -85,B 0,C 180,E1 -14931.402,E2 -14931.402} C_VEL
LIN {X 0,Y 327.888,Z 477.338,A -85,B 0,C 180,E1 -14933.23,E2 -14933.23} C_VEL
LIN {X 0,Y 326.796,Z 479.686,A -85,B 0,C 180,E1 -14935.065,E2 -14935.065} C_VEL
LIN {X 0,Y 326.245,Z 480.462,A -85,B 0,C 180,E1 -14936.295,E2 -14936.295} C_VEL
LIN {X 0,Y 325.89,Z 480.594,A -85,B 0,C 180,E1 -14937.528,E2 -14937.528} C_VEL
LIN {X 0,Y 325.694,Z 480.079,A -85,B 0,C 180,E1 -14938.764,E2 -14938.764} C_VEL
LIN {X 0,Y 325.567,Z 478.921,A -85,B 0,C 180,E1 -14940,E2 -14940} C_VEL
LIN {X 0,Y 325.523,Z 475.943,A -85,B 0,C 180,E1 -14941.856,E2 -14941.856} C_VEL
LIN {X 0,Y 325.68,Z 471.363,A -85,B 0,C 180,E1 -14943.712,E2 -14943.712} C_VEL
LIN {X 0,Y 326.006,Z 466.124,A -85,B 0,C 180,E1 -14945.257,E2 -14945.257} C_VEL
LIN {X 0,Y 326.298,Z 459.384,A -85,B 0,C 180,E1 -14946.803,E2 -14946.803} C_VEL
LIN {X 0,Y 326.622,Z 450.549,A -85,B 0,C 180,E1 -14948.379,E2 -14948.379} C_VEL
LIN {X 0,Y 326.99,Z 441.907,A -85,B 0,C 180,E1 -14949.589,E2 -14949.589} C_VEL
LIN {X 0,Y 327.488,Z 432.147,A -85,B 0,C 180,E1 -14950.667,E2 -14950.667} C_VEL
LIN {X 0,Y 327.179,Z 426.99,A -85,B 0,C 180,E1 -14951.147,E2 -14951.147} C_VEL
LIN {X 0,Y 325.938,Z 416.124,A -85,B 0,C 180,E1 -14951.978,E2 -14951.978} C_VEL
LIN {X 0,Y 325.557,Z 412.173,A -85,B 0,C 180,E1 -14952.23,E2 -14952.23} C_VEL
LIN {X 0,Y 325.696,Z 406.242,A -85,B 0,C 180,E1 -14955.648,E2 -14955.648} C_VEL
LIN {X 0,Y 325.925,Z 400.752,A -85,B 0,C 180,E1 -14958.872,E2 -14958.872} C_VEL
LIN {X 0,Y 326.253,Z 394.169,A -85,B 0,C 180,E1 -14962.815,E2 -14962.815} C_VEL
LIN {X 0,Y 326.621,Z 387.546,A -85,B 0,C 180,E1 -14966.863,E2 -14966.863} C_VEL
LIN {X 0,Y 326.979,Z 383.115,A -85,B 0,C 180,E1 -14969.628,E2 -14969.628} C_VEL
LIN {X 0,Y 326.807,Z 379.776,A -85,B 0,C 180,E1 -14971.795,E2 -14971.795} C_VEL
LIN {X 0,Y 326.619,Z 379.798,A -85,B 0,C 180,E1 -14975.519,E2 -14975.519} C_VEL
LIN {X 0,Y 326.614,Z 379.8,A -85,B 0,C 180,E1 -14979.227,E2 -14979.227} C_VEL
LIN {X 0,Y 326.585,Z 379.805,A -85,B 0,C 180,E1 -14982.973,E2 -14982.973} C_VEL
LIN {X 0,Y 326.585,Z 379.804,A -85,B 0,C 180,E1 -14987.027,E2 -14987.027} C_VEL
LIN {X 0,Y 326.614,Z 379.802,A -85,B 0,C 180,E1 -14990.773,E2 -14990.773} C_VEL
LIN {X 0,Y 326.616,Z 379.802,A -85,B 0,C 180,E1 -14994.48,E2 -14994.48} C_VEL
LIN {X 0,Y 326.61,Z 379.798,A -85,B 0,C 180,E1 -14997.456,E2 -14997.456} C_VEL
LIN {X 0,Y 326.651,Z 379.797,A -85,B 0,C 180,E1 -15000.34,E2 -15000.34} C_VEL
LIN {X 0,Y 326.693,Z 379.793,A -85,B 0,C 180,E1 -15004.516,E2 -15004.516} C_VEL
LIN {X 0,Y 326.65,Z 379.797,A -85,B 0,C 180,E1 -15008.545,E2 -15008.545} C_VEL
LIN {X 0,Y 326.747,Z 379.781,A -85,B 0,C 180,E1 -15011.177,E2 -15011.177} C_VEL
LIN {X 0,Y 326.766,Z 379.779,A -85,B 0,C 180,E1 -15015.433,E2 -15015.433} C_VEL
LIN {X 0,Y 326.773,Z 379.778,A -85,B 0,C 180,E1 -15018.839,E2 -15018.839} C_VEL
LIN {X 0,Y 326.961,Z 379.756,A -85,B 0,C 180,E1 -15022.59,E2 -15022.59} C_VEL
LIN {X 0,Y 326.779,Z 379.777,A -85,B 0,C 180,E1 -15025.065,E2 -15025.065} C_VEL
LIN {X 0,Y 327.049,Z 379.745,A -85,B 0,C 180,E1 -15027.537,E2 -15027.537} C_VEL
LIN {X 0,Y 327.201,Z 379.73,A -85,B 0,C 180,E1 -15030,E2 -15030} C_VEL
LIN {X 0,Y 327.051,Z 379.745,A -85,B 0,C 180,E1 -15032.463,E2 -15032.463} C_VEL
LIN {X 0,Y 326.993,Z 379.753,A -85,B 0,C 180,E1 -15036.169,E2 -15036.169} C_VEL
LIN {X 0,Y 326.918,Z 379.76,A -85,B 0,C 180,E1 -15038.655,E2 -15038.655} C_VEL
LIN {X 0,Y 326.738,Z 379.783,A -85,B 0,C 180,E1 -15042.421,E2 -15042.421} C_VEL
LIN {X 0,Y 326.757,Z 379.78,A -85,B 0,C 180,E1 -15044.957,E2 -15044.957} C_VEL
LIN {X 0,Y 326.738,Z 379.782,A -85,B 0,C 180,E1 -15048.84,E2 -15048.84} C_VEL
LIN {X 0,Y 326.624,Z 379.796,A -85,B 0,C 180,E1 -15052.787,E2 -15052.787} C_VEL
LIN {X 0,Y 326.692,Z 379.793,A -85,B 0,C 180,E1 -15055.484,E2 -15055.484} C_VEL
LIN {X 0,Y 326.65,Z 379.797,A -85,B 0,C 180,E1 -15059.66,E2 -15059.66} C_VEL
LIN {X 0,Y 326.609,Z 379.799,A -85,B 0,C 180,E1 -15064.019,E2 -15064.019} C_VEL
LIN {X 0,Y 326.631,Z 379.8,A -85,B 0,C 180,E1 -15067.239,E2 -15067.239} C_VEL
LIN {X 0,Y 326.58,Z 379.806,A -85,B 0,C 180,E1 -15071.131,E2 -15071.131} C_VEL
LIN {X 0,Y 326.529,Z 379.809,A -85,B 0,C 180,E1 -15074.743,E2 -15074.743} C_VEL
LIN {X 0,Y 326.578,Z 379.802,A -85,B 0,C 180,E1 -15078.154,E2 -15078.154} C_VEL
LIN {X 0,Y 326.599,Z 379.803,A -85,B 0,C 180,E1 -15081.388,E2 -15081.388} C_VEL
LIN {X 0,Y 326.621,Z 379.8,A -85,B 0,C 180,E1 -15084.851,E2 -15084.851} C_VEL
LIN {X 0,Y 326.609,Z 379.8,A -85,B 0,C 180,E1 -15087.455,E2 -15087.455} C_VEL
LIN {X 0,Y 326.662,Z 379.792,A -85,B 0,C 180,E1 -15090.341,E2 -15090.341} C_VEL
LIN {X 0,Y 326.692,Z 379.79,A -85,B 0,C 180,E1 -15094.516,E2 -15094.516} C_VEL
LIN {X 0,Y 326.65,Z 379.796,A -85,B 0,C 180,E1 -15098.545,E2 -15098.545} C_VEL
LIN {X 0,Y 326.746,Z 379.783,A -85,B 0,C 180,E1 -15101.177,E2 -15101.177} C_VEL
LIN {X 0,Y 326.724,Z 379.783,A -85,B 0,C 180,E1 -15104.44,E2 -15104.44} C_VEL
LIN {X 0,Y 326.085,Z 379.866,A -85,B 0,C 180,E1 -15105.468,E2 -15105.468} C_VEL
LIN {X 0,Y 323.264,Z 380.222,A -85,B 0,C 180,E1 -15107.142,E2 -15107.142} C_VEL
LIN {X 0,Y 320.864,Z 380.52,A -85,B 0,C 180,E1 -15108.498,E2 -15108.498} C_VEL
LIN {X 0,Y 319.841,Z 380.643,A -85,B 0,C 180,E1 -15109.548,E2 -15109.548} C_VEL
LIN {X 0,Y 319.762,Z 380.651,A -85,B 0,C 180,E1 -15109.904,E2 -15109.904} C_VEL
LIN {X 0,Y 319.936,Z 380.633,A -85,B 0,C 180,E1 -15112.426,E2 -15112.426} C_VEL
LIN {X 0,Y 319.749,Z 380.655,A -85,B 0,C 180,E1 -15114.956,E2 -15114.956} C_VEL
LIN {X 0,Y 319.992,Z 380.622,A -85,B 0,C 180,E1 -15117.482,E2 -15117.482} C_VEL
LIN {X 0,Y 320.153,Z 380.604,A -85,B 0,C 180,E1 -15120,E2 -15120} C_VEL
LIN {X 0,Y 320.011,Z 380.625,A -85,B 0,C 180,E1 -15122.517,E2 -15122.517} C_VEL
LIN {X 0,Y 319.954,Z 380.632,A -85,B 0,C 180,E1 -15126.305,E2 -15126.305} C_VEL
LIN {X 0,Y 319.844,Z 380.642,A -85,B 0,C 180,E1 -15128.848,E2 -15128.848} C_VEL
LIN {X 0,Y 319.684,Z 380.663,A -85,B 0,C 180,E1 -15132.7,E2 -15132.7} C_VEL
LIN {X 0,Y 319.701,Z 380.659,A -85,B 0,C 180,E1 -15135.295,E2 -15135.295} C_VEL
LIN {X 0,Y 319.676,Z 380.662,A -85,B 0,C 180,E1 -15139.255,E2 -15139.255} C_VEL
LIN {X 0,Y 319.572,Z 380.675,A -85,B 0,C 180,E1 -15143.319,E2 -15143.319} C_VEL
LIN {X 0,Y 319.635,Z 380.672,A -85,B 0,C 180,E1 -15146.088,E2 -15146.088} C_VEL
LIN {X 0,Y 319.581,Z 380.674,A -85,B 0,C 180,E1 -15148.934,E2 -15148.934} C_VEL
LIN {X 0,Y 319.533,Z 380.684,A -85,B 0,C 180,E1 -15151.862,E2 -15151.862} C_VEL
LIN {X 0,Y 319.581,Z 380.676,A -85,B 0,C 180,E1 -15155.543,E2 -15155.543} C_VEL
LIN {X 0,Y 319.575,Z 380.679,A -85,B 0,C 180,E1 -15158.008,E2 -15158.008} C_VEL
LIN {X 0,Y 319.53,Z 380.683,A -85,B 0,C 180,E1 -15161.598,E2 -15161.598} C_VEL
LIN {X 0,Y 319.547,Z 380.679,A -85,B 0,C 180,E1 -15165.268,E2 -15165.268} C_VEL
LIN {X 0,Y 319.534,Z 380.679,A -85,B 0,C 180,E1 -15168.713,E2 -15168.713} C_VEL
LIN {X 0,Y 319.597,Z 380.705,A -85,B 0,C 180,E1 -15170.072,E2 -15170.072} C_VEL
LIN {X 0,Y 321.252,Z 389.043,A -85,B 0,C 180,E1 -15173.406,E2 -15173.406} C_VEL
LIN {X 0,Y 323.248,Z 398.622,A -85,B 0,C 180,E1 -15177.075,E2 -15177.075} C_VEL
LIN {X 0,Y 324.516,Z 404.94,A -85,B 0,C 180,E1 -15179.408,E2 -15179.408} C_VEL
LIN {X 0,Y 323.632,Z 410.953,A -85,B 0,C 180,E1 -15181.461,E2 -15181.461} C_VEL
LIN {X 0,Y 321.697,Z 422.795,A -85,B 0,C 180,E1 -15185.475,E2 -15185.475} C_VEL
LIN {X 0,Y 319.983,Z 436.511,A -85,B 0,C 180,E1 -15190.097,E2 -15190.097} C_VEL
LIN {X 0,Y 319.636,Z 440.114,A -85,B 0,C 180,E1 -15191.307,E2 -15191.307} C_VEL
LIN {X 0,Y 320.249,Z 452.43,A -85,B 0,C 180,E1 -15191.841,E2 -15191.841} C_VEL
LIN {X 0,Y 321.155,Z 465.262,A -85,B 0,C 180,E1 -15192.653,E2 -15192.653} C_VEL
LIN {X 0,Y 321.538,Z 473.579,A -85,B 0,C 180,E1 -15193.329,E2 -15193.329} C_VEL
LIN {X 0,Y 320.843,Z 484.584,A -85,B 0,C 180,E1 -15194.436,E2 -15194.436} C_VEL
LIN {X 0,Y 320.079,Z 494.603,A -85,B 0,C 180,E1 -15195.699,E2 -15195.699} C_VEL
LIN {X 0,Y 319.572,Z 502.876,A -85,B 0,C 180,E1 -15196.973,E2 -15196.973} C_VEL
LIN {X 0,Y 319.016,Z 511.376,A -85,B 0,C 180,E1 -15198.564,E2 -15198.564} C_VEL
LIN {X 0,Y 318.611,Z 519.523,A -85,B 0,C 180,E1 -15200.477,E2 -15200.477} C_VEL
LIN {X 0,Y 318.484,Z 525.982,A -85,B 0,C 180,E1 -15202.392,E2 -15202.392} C_VEL
LIN {X 0,Y 318.499,Z 530.942,A -85,B 0,C 180,E1 -15204.301,E2 -15204.301} C_VEL
LIN {X 0,Y 318.516,Z 534.624,A -85,B 0,C 180,E1 -15206.205,E2 -15206.205} C_VEL
LIN {X 0,Y 318.66,Z 536.464,A -85,B 0,C 180,E1 -15207.472,E2 -15207.472} C_VEL
LIN {X 0,Y 318.577,Z 537.766,A -85,B 0,C 180,E1 -15208.736,E2 -15208.736} C_VEL
LIN {X 0,Y 318.526,Z 538.606,A -85,B 0,C 180,E1 -15210,E2 -15210} C_VEL
LIN {X 0,Y 318.551,Z 539.032,A -85,B 0,C 180,E1 -15211.264,E2 -15211.264} C_VEL
LIN {X 0,Y 318.404,Z 538.967,A -85,B 0,C 180,E1 -15212.53,E2 -15212.53} C_VEL
LIN {X 0,Y 318.15,Z 537.564,A -85,B 0,C 180,E1 -15215.069,E2 -15215.069} C_VEL
LIN {X 0,Y 318.123,Z 536.208,A -85,B 0,C 180,E1 -15216.342,E2 -15216.342} C_VEL
LIN {X 0,Y 318.196,Z 533.361,A -85,B 0,C 180,E1 -15218.254,E2 -15218.254} C_VEL
LIN {X 0,Y 318.496,Z 529.492,A -85,B 0,C 180,E1 -15220.168,E2 -15220.168} C_VEL
LIN {X 0,Y 319.175,Z 524.511,A -85,B 0,C 180,E1 -15222.075,E2 -15222.075} C_VEL
LIN {X 0,Y 320.278,Z 518.318,A -85,B 0,C 180,E1 -15223.968,E2 -15223.968} C_VEL
LIN {X 0,Y 321.522,Z 511.327,A -85,B 0,C 180,E1 -15225.706,E2 -15225.706} C_VEL
LIN {X 0,Y 323.214,Z 502.936,A -85,B 0,C 180,E1 -15227.397,E2 -15227.397} C_VEL
LIN {X 0,Y 325.269,Z 492.629,A -85,B 0,C 180,E1 -15229.075,E2 -15229.075} C_VEL
LIN {X 0,Y 327.431,Z 480.9,A -85,B 0,C 180,E1 -15230.578,E2 -15230.578} C_VEL
LIN {X 0,Y 328.307,Z 469.457,A -85,B 0,C 180,E1 -15231.838,E2 -15231.838} C_VEL
LIN {X 0,Y 327.959,Z 459.272,A -85,B 0,C 180,E1 -15232.858,E2 -15232.858} C_VEL
LIN {X 0,Y 325.957,Z 446.231,A -85,B 0,C 180,E1 -15234.114,E2 -15234.114} C_VEL
LIN {X 0,Y 323.829,Z 437.068,A -85,B 0,C 180,E1 -15234.967,E2 -15234.967} C_VEL
LIN {X 0,Y 326.649,Z 427.067,A -85,B 0,C 180,E1 -15238.954,E2 -15238.954} C_VEL
LIN {X 0,Y 328.384,Z 422.089,A -85,B 0,C 180,E1 -15241.122,E2 -15241.122} C_VEL
LIN {X 0,Y 328.8,Z 419.746,A -85,B 0,C 180,E1 -15242.301,E2 -15242.301} C_VEL
LIN {X 0,Y 328.294,Z 416.061,A -85,B 0,C 180,E1 -15244.563,E2 -15244.563} C_VEL
LIN {X 0,Y 327.393,Z 412.3,A -85,B 0,C 180,E1 -15247.414,E2 -15247.414} C_VEL
LIN {X 0,Y 326.771,Z 409.375,A -85,B 0,C 180,E1 -15250.183,E2 -15250.183} C_VEL
LIN {X 0,Y 326.137,Z 406.838,A -85,B 0,C 180,E1 -15253.597,E2 -15253.597} C_VEL
LIN {X 0,Y 325.785,Z 405.623,A -85,B 0,C 180,E1 -15256.344,E2 -15256.344} C_VEL
LIN {X 0,Y 325.448,Z 405.064,A -85,B 0,C 180,E1 -15259.621,E2 -15259.621} C_VEL
LIN {X 0,Y 325.222,Z 405.442,A -85,B 0,C 180,E1 -15263.089,E2 -15263.089} C_VEL
LIN {X 0,Y 325.141,Z 406.358,A -85,B 0,C 180,E1 -15265.806,E2 -15265.806} C_VEL
LIN {X 0,Y 324.765,Z 408.009,A -85,B 0,C 180,E1 -15268.71,E2 -15268.71} C_VEL
LIN {X 0,Y 324.037,Z 410.185,A -85,B 0,C 180,E1 -15271.5,E2 -15271.5} C_VEL
LIN {X 0,Y 323.211,Z 412.715,A -85,B 0,C 180,E1 -15274.222,E2 -15274.222} C_VEL
LIN {X 0,Y 322.177,Z 416.956,A -85,B 0,C 180,E1 -15278.233,E2 -15278.233} C_VEL
LIN {X 0,Y 321.798,Z 419.443,A -85,B 0,C 180,E1 -15280.273,E2 -15280.273} C_VEL
LIN {X 0,Y 325.807,Z 431.05,A -85,B 0,C 180,E1 -15282.098,E2 -15282.098} C_VEL
LIN {X 0,Y 328.037,Z 440.73,A -85,B 0,C 180,E1 -15283.665,E2 -15283.665} C_VEL
LIN {X 0,Y 328.726,Z 447.411,A -85,B 0,C 180,E1 -15284.793,E2 -15284.793} C_VEL
LIN {X 0,Y 326.948,Z 456.719,A -85,B 0,C 180,E1 -15286.323,E2 -15286.323} C_VEL
LIN {X 0,Y 325.236,Z 464.039,A -85,B 0,C 180,E1 -15287.837,E2 -15287.837} C_VEL
LIN {X 0,Y 323.729,Z 469.794,A -85,B 0,C 180,E1 -15289.366,E2 -15289.366} C_VEL
LIN {X 0,Y 322.206,Z 474.971,A -85,B 0,C 180,E1 -15291.217,E2 -15291.217} C_VEL
LIN {X 0,Y 321.254,Z 477.574,A -85,B 0,C 180,E1 -15292.458,E2 -15292.458} C_VEL
LIN {X 0,Y 320.472,Z 479.485,A -85,B 0,C 180,E1 -15293.705,E2 -15293.705} C_VEL
LIN {X 0,Y 319.801,Z 480.743,A -85,B 0,C 180,E1 -15294.957,E2 -15294.957} C_VEL
LIN {X 0,Y 319.219,Z 481.364,A -85,B 0,C 180,E1 -15296.213,E2 -15296.213} C_VEL
LIN {X 0,Y 318.854,Z 481.344,A -85,B 0,C 180,E1 -15297.474,E2 -15297.474} C_VEL
LIN {X 0,Y 318.651,Z 480.692,A -85,B 0,C 180,E1 -15298.736,E2 -15298.736} C_VEL
LIN {X 0,Y 318.492,Z 479.405,A -85,B 0,C 180,E1 -15300,E2 -15300} C_VEL
LIN {X 0,Y 318.455,Z 476.223,A -85,B 0,C 180,E1 -15301.897,E2 -15301.897} C_VEL
LIN {X 0,Y 318.598,Z 471.427,A -85,B 0,C 180,E1 -15303.795,E2 -15303.795} C_VEL
LIN {X 0,Y 318.939,Z 466.045,A -85,B 0,C 180,E1 -15305.374,E2 -15305.374} C_VEL
LIN {X 0,Y 319.239,Z 459.123,A -85,B 0,C 180,E1 -15306.955,E2 -15306.955} C_VEL
LIN {X 0,Y 319.563,Z 450.451,A -85,B 0,C 180,E1 -15308.492,E2 -15308.492} C_VEL
LIN {X 0,Y 319.974,Z 441.038,A -85,B 0,C 180,E1 -15309.801,E2 -15309.801} C_VEL
LIN {X 0,Y 320.481,Z 430.902,A -85,B 0,C 180,E1 -15310.903,E2 -15310.903} C_VEL
LIN {X 0,Y 319.231,Z 420.116,A -85,B 0,C 180,E1 -15311.831,E2 -15311.831} C_VEL
LIN {X 0,Y 318.488,Z 412.485,A -85,B 0,C 180,E1 -15312.344,E2 -15312.344} C_VEL
LIN {X 0,Y 318.65,Z 406.243,A -85,B 0,C 180,E1 -15316.004,E2 -15316.004} C_VEL
LIN {X 0,Y 318.99,Z 399.602,A -85,B 0,C 180,E1 -15319.968,E2 -15319.968} C_VEL
LIN {X 0,Y 319.292,Z 392.966,A -85,B 0,C 180,E1 -15324.03,E2 -15324.03} C_VEL
LIN {X 0,Y 319.648,Z 387.396,A -85,B 0,C 180,E1 -15327.498,E2 -15327.498} C_VEL
LIN {X 0,Y 319.921,Z 382.913,A -85,B 0,C 180,E1 -15330.349,E2 -15330.349} C_VEL
LIN {X 0,Y 319.765,Z 380.653,A -85,B 0,C 180,E1 -15331.836,E2 -15331.836} C_VEL
LIN {X 0,Y 319.563,Z 380.677,A -85,B 0,C 180,E1 -15336.427,E2 -15336.427} C_VEL
LIN {X 0,Y 319.561,Z 380.676,A -85,B 0,C 180,E1 -15339.669,E2 -15339.669} C_VEL
LIN {X 0,Y 319.56,Z 380.677,A -85,B 0,C 180,E1 -15343.467,E2 -15343.467} C_VEL
LIN {X 0,Y 319.563,Z 380.679,A -85,B 0,C 180,E1 -15347.018,E2 -15347.018} C_VEL
LIN {X 0,Y 319.55,Z 380.68,A -85,B 0,C 180,E1 -15350.371,E2 -15350.371} C_VEL
LIN {X 0,Y 319.583,Z 380.678,A -85,B 0,C 180,E1 -15354.457,E2 -15354.457} C_VEL
LIN {X 0,Y 319.533,Z 380.682,A -85,B 0,C 180,E1 -15358.138,E2 -15358.138} C_VEL
LIN {X 0,Y 319.614,Z 380.669,A -85,B 0,C 180,E1 -15361.59,E2 -15361.59} C_VEL
LIN {X 0,Y 319.608,Z 380.67,A -85,B 0,C 180,E1 -15365.304,E2 -15365.304} C_VEL
LIN {X 0,Y 319.6,Z 380.674,A -85,B 0,C 180,E1 -15368.048,E2 -15368.048} C_VEL
LIN {X 0,Y 319.692,Z 380.66,A -85,B 0,C 180,E1 -15370.962,E2 -15370.962} C_VEL
LIN {X 0,Y 319.734,Z 380.654,A -85,B 0,C 180,E1 -15375.276,E2 -15375.276} C_VEL
LIN {X 0,Y 319.756,Z 380.655,A -85,B 0,C 180,E1 -15379.873,E2 -15379.873} C_VEL
LIN {X 0,Y 319.916,Z 380.635,A -85,B 0,C 180,E1 -15382.426,E2 -15382.426} C_VEL
LIN {X 0,Y 319.748,Z 380.653,A -85,B 0,C 180,E1 -15384.956,E2 -15384.956} C_VEL
LIN {X 0,Y 319.993,Z 380.623,A -85,B 0,C 180,E1 -15387.482,E2 -15387.482} C_VEL
LIN {X 0,Y 320.153,Z 380.608,A -85,B 0,C 180,E1 -15390,E2 -15390} C_VEL
LIN {X 0,Y 319.995,Z 380.623,A -85,B 0,C 180,E1 -15392.517,E2 -15392.517} C_VEL
LIN {X 0,Y 319.948,Z 380.63,A -85,B 0,C 180,E1 -15396.305,E2 -15396.305} C_VEL
LIN {X 0,Y 319.845,Z 380.641,A -85,B 0,C 180,E1 -15398.848,E2 -15398.848} C_VEL
LIN {X 0,Y 319.685,Z 380.66,A -85,B 0,C 180,E1 -15402.7,E2 -15402.7} C_VEL
LIN {X 0,Y 319.702,Z 380.66,A -85,B 0,C 180,E1 -15405.295,E2 -15405.295} C_VEL
LIN {X 0,Y 319.68,Z 380.663,A -85,B 0,C 180,E1 -15409.255,E2 -15409.255} C_VEL
LIN {X 0,Y 319.574,Z 380.677,A -85,B 0,C 180,E1 -15413.319,E2 -15413.319} C_VEL
LIN {X 0,Y 319.637,Z 380.668,A -85,B 0,C 180,E1 -15416.088,E2 -15416.088} C_VEL
LIN {X 0,Y 319.582,Z 380.674,A -85,B 0,C 180,E1 -15418.934,E2 -15418.934} C_VEL
LIN {X 0,Y 319.533,Z 380.682,A -85,B 0,C 180,E1 -15421.862,E2 -15421.862} C_VEL
LIN {X 0,Y 319.583,Z 380.678,A -85,B 0,C 180,E1 -15425.543,E2 -15425.543} C_VEL
LIN {X 0,Y 319.576,Z 380.675,A -85,B 0,C 180,E1 -15428.008,E2 -15428.008} C_VEL
LIN {X 0,Y 319.528,Z 380.683,A -85,B 0,C 180,E1 -15431.597,E2 -15431.597} C_VEL
LIN {X 0,Y 319.49,Z 380.69,A -85,B 0,C 180,E1 -15435.257,E2 -15435.257} C_VEL
LIN {X 0,Y 319.53,Z 380.681,A -85,B 0,C 180,E1 -15438.712,E2 -15438.712} C_VEL
LIN {X 0,Y 319.556,Z 380.677,A -85,B 0,C 180,E1 -15442.349,E2 -15442.349} C_VEL
LIN {X 0,Y 319.562,Z 380.681,A -85,B 0,C 180,E1 -15445.123,E2 -15445.123} C_VEL
LIN {X 0,Y 319.572,Z 380.68,A -85,B 0,C 180,E1 -15449.058,E2 -15449.058} C_VEL
LIN {X 0,Y 319.61,Z 380.671,A -85,B 0,C 180,E1 -15452.498,E2 -15452.498} C_VEL
LIN {X 0,Y 319.607,Z 380.672,A -85,B 0,C 180,E1 -15455.304,E2 -15455.304} C_VEL
LIN {X 0,Y 319.6,Z 380.671,A -85,B 0,C 180,E1 -15458.048,E2 -15458.048} C_VEL
LIN {X 0,Y 319.691,Z 380.664,A -85,B 0,C 180,E1 -15460.962,E2 -15460.962} C_VEL
LIN {X 0,Y 319.733,Z 380.656,A -85,B 0,C 180,E1 -15465.276,E2 -15465.276} C_VEL
LIN {X 0,Y 319.762,Z 380.651,A -85,B 0,C 180,E1 -15469.904,E2 -15469.904} C_VEL
LIN {X 0,Y 319.105,Z 380.735,A -85,B 0,C 180,E1 -15470.958,E2 -15470.958} C_VEL
LIN {X 0,Y 316.251,Z 381.094,A -85,B 0,C 180,E1 -15472.673,E2 -15472.673} C_VEL
LIN {X 0,Y 313.821,Z 381.395,A -85,B 0,C 180,E1 -15474.063,E2 -15474.063} C_VEL
LIN {X 0,Y 312.774,Z 381.523,A -85,B 0,C 180,E1 -15475.14,E2 -15475.14} C_VEL
LIN {X 0,Y 312.687,Z 381.532,A -85,B 0,C 180,E1 -15475.505,E2 -15475.505} C_VEL
LIN {X 0,Y 312.993,Z 381.498,A -85,B 0,C 180,E1 -15478.713,E2 -15478.713} C_VEL
LIN {X 0,Y 312.995,Z 381.494,A -85,B 0,C 180,E1 -15481.287,E2 -15481.287} C_VEL
LIN {X 0,Y 312.698,Z 381.532,A -85,B 0,C 180,E1 -15483.866,E2 -15483.866} C_VEL
LIN {X 0,Y 312.912,Z 381.509,A -85,B 0,C 180,E1 -15486.448,E2 -15486.448} C_VEL
LIN {X 0,Y 312.789,Z 381.52,A -85,B 0,C 180,E1 -15489.049,E2 -15489.049} C_VEL
LIN {X 0,Y 312.636,Z 381.539,A -85,B 0,C 180,E1 -15492.991,E2 -15492.991} C_VEL
LIN {X 0,Y 312.64,Z 381.539,A -85,B 0,C 180,E1 -15495.65,E2 -15495.65} C_VEL
LIN {X 0,Y 312.632,Z 381.539,A -85,B 0,C 180,E1 -15499.237,E2 -15499.237} C_VEL
LIN {X 0,Y 312.547,Z 381.55,A -85,B 0,C 180,E1 -15502.789,E2 -15502.789} C_VEL
LIN {X 0,Y 312.604,Z 381.547,A -85,B 0,C 180,E1 -15505.935,E2 -15505.935} C_VEL
LIN {X 0,Y 312.539,Z 381.553,A -85,B 0,C 180,E1 -15509.651,E2 -15509.651} C_VEL
LIN {X 0,Y 312.521,Z 381.556,A -85,B 0,C 180,E1 -15513.689,E2 -15513.689} C_VEL
LIN {X 0,Y 312.539,Z 381.552,A -85,B 0,C 180,E1 -15517.383,E2 -15517.383} C_VEL
LIN {X 0,Y 312.493,Z 381.556,A -85,B 0,C 180,E1 -15520.709,E2 -15520.709} C_VEL
LIN {X 0,Y 312.476,Z 381.56,A -85,B 0,C 180,E1 -15524.205,E2 -15524.205} C_VEL
LIN {X 0,Y 312.522,Z 381.556,A -85,B 0,C 180,E1 -15527.911,E2 -15527.911} C_VEL
LIN {X 0,Y 312.544,Z 381.571,A -85,B 0,C 180,E1 -15529.724,E2 -15529.724} C_VEL
LIN {X 0,Y 314.067,Z 389.117,A -85,B 0,C 180,E1 -15532.829,E2 -15532.829} C_VEL
LIN {X 0,Y 316.22,Z 399.559,A -85,B 0,C 180,E1 -15536.947,E2 -15536.947} C_VEL
LIN {X 0,Y 317.47,Z 406.011,A -85,B 0,C 180,E1 -15539.392,E2 -15539.392} C_VEL
LIN {X 0,Y 316.16,Z 413.973,A -85,B 0,C 180,E1 -15542.172,E2 -15542.172} C_VEL
LIN {X 0,Y 314.134,Z 426.47,A -85,B 0,C 180,E1 -15546.532,E2 -15546.532} C_VEL
LIN {X 0,Y 312.592,Z 439.775,A -85,B 0,C 180,E1 -15551.142,E2 -15551.142} C_VEL
LIN {X 0,Y 313.204,Z 453.334,A -85,B 0,C 180,E1 -15551.775,E2 -15551.775} C_VEL
LIN {X 0,Y 314.057,Z 465.423,A -85,B 0,C 180,E1 -15552.584,E2 -15552.584} C_VEL
LIN {X 0,Y 314.439,Z 473.632,A -85,B 0,C 180,E1 -15553.276,E2 -15553.276} C_VEL
LIN {X 0,Y 313.679,Z 485.586,A -85,B 0,C 180,E1 -15554.537,E2 -15554.537} C_VEL
LIN {X 0,Y 312.895,Z 495.527,A -85,B 0,C 180,E1 -15555.862,E2 -15555.862} C_VEL
LIN {X 0,Y 312.356,Z 504.41,A -85,B 0,C 180,E1 -15557.328,E2 -15557.328} C_VEL
LIN {X 0,Y 311.844,Z 512.472,A -85,B 0,C 180,E1 -15558.956,E2 -15558.956} C_VEL
LIN {X 0,Y 311.532,Z 520.277,A -85,B 0,C 180,E1 -15560.914,E2 -15560.914} C_VEL
LIN {X 0,Y 311.467,Z 527.095,A -85,B 0,C 180,E1 -15563.133,E2 -15563.133} C_VEL
LIN {X 0,Y 311.466,Z 531.068,A -85,B 0,C 180,E1 -15564.822,E2 -15564.822} C_VEL
LIN {X 0,Y 311.471,Z 533.491,A -85,B 0,C 180,E1 -15566.119,E2 -15566.119} C_VEL
LIN {X 0,Y 311.615,Z 535.392,A -85,B 0,C 180,E1 -15567.415,E2 -15567.415} C_VEL
LIN {X 0,Y 311.537,Z 536.804,A -85,B 0,C 180,E1 -15568.707,E2 -15568.707} C_VEL
LIN {X 0,Y 311.485,Z 537.712,A -85,B 0,C 180,E1 -15570,E2 -15570} C_VEL
LIN {X 0,Y 311.504,Z 538.192,A -85,B 0,C 180,E1 -15571.293,E2 -15571.293} C_VEL
LIN {X 0,Y 311.335,Z 538.228,A -85,B 0,C 180,E1 -15572.588,E2 -15572.588} C_VEL
LIN {X 0,Y 311.125,Z 537.787,A -85,B 0,C 180,E1 -15573.886,E2 -15573.886} C_VEL
LIN {X 0,Y 311.046,Z 536.002,A -85,B 0,C 180,E1 -15576.19,E2 -15576.19} C_VEL
LIN {X 0,Y 311.12,Z 532.976,A -85,B 0,C 180,E1 -15578.443,E2 -15578.443} C_VEL
LIN {X 0,Y 311.471,Z 529.252,A -85,B 0,C 180,E1 -15580.4,E2 -15580.4} C_VEL
LIN {X 0,Y 312.212,Z 524.434,A -85,B 0,C 180,E1 -15582.348,E2 -15582.348} C_VEL
LIN {X 0,Y 313.585,Z 517.294,A -85,B 0,C 180,E1 -15584.604,E2 -15584.604} C_VEL
LIN {X 0,Y 315.072,Z 510.024,A -85,B 0,C 180,E1 -15586.431,E2 -15586.431} C_VEL
LIN {X 0,Y 316.86,Z 501.885,A -85,B 0,C 180,E1 -15588.091,E2 -15588.091} C_VEL
LIN {X 0,Y 319.071,Z 491.59,A -85,B 0,C 180,E1 -15589.795,E2 -15589.795} C_VEL
LIN {X 0,Y 321.274,Z 479.913,A -85,B 0,C 180,E1 -15591.326,E2 -15591.326} C_VEL
LIN {X 0,Y 322.148,Z 468.726,A -85,B 0,C 180,E1 -15592.603,E2 -15592.603} C_VEL
LIN {X 0,Y 321.489,Z 457.17,A -85,B 0,C 180,E1 -15593.842,E2 -15593.842} C_VEL
LIN {X 0,Y 319.658,Z 445.887,A -85,B 0,C 180,E1 -15595.008,E2 -15595.008} C_VEL
LIN {X 0,Y 317.487,Z 436.569,A -85,B 0,C 180,E1 -15595.96,E2 -15595.96} C_VEL
LIN {X 0,Y 320.214,Z 427.882,A -85,B 0,C 180,E1 -15599.593,E2 -15599.593} C_VEL
LIN {X 0,Y 321.834,Z 423.443,A -85,B 0,C 180,E1 -15601.608,E2 -15601.608} C_VEL
LIN {X 0,Y 321.927,Z 420.8,A -85,B 0,C 180,E1 -15603.078,E2 -15603.078} C_VEL
LIN {X 0,Y 321.609,Z 418.402,A -85,B 0,C 180,E1 -15604.623,E2 -15604.623} C_VEL
LIN {X 0,Y 320.636,Z 414.26,A -85,B 0,C 180,E1 -15607.9,E2 -15607.9} C_VEL
LIN {X 0,Y 319.968,Z 411.063,A -85,B 0,C 180,E1 -15611.219,E2 -15611.219} C_VEL
LIN {X 0,Y 319.364,Z 408.824,A -85,B 0,C 180,E1 -15614.765,E2 -15614.765} C_VEL
LIN {X 0,Y 319.087,Z 408.007,A -85,B 0,C 180,E1 -15616.938,E2 -15616.938} C_VEL
LIN {X 0,Y 318.739,Z 407.565,A -85,B 0,C 180,E1 -15620.51,E2 -15620.51} C_VEL
LIN {X 0,Y 318.536,Z 407.959,A -85,B 0,C 180,E1 -15623.436,E2 -15623.436} C_VEL
LIN {X 0,Y 318.326,Z 409.051,A -85,B 0,C 180,E1 -15626.499,E2 -15626.499} C_VEL
LIN {X 0,Y 317.808,Z 410.894,A -85,B 0,C 180,E1 -15629.593,E2 -15629.593} C_VEL
LIN {X 0,Y 316.916,Z 413.239,A -85,B 0,C 180,E1 -15632.505,E2 -15632.505} C_VEL
LIN {X 0,Y 315.764,Z 416.954,A -85,B 0,C 180,E1 -15636.383,E2 -15636.383} C_VEL
LIN {X 0,Y 315.161,Z 420.146,A -85,B 0,C 180,E1 -15639.195,E2 -15639.195} C_VEL
LIN {X 0,Y 315.795,Z 422.189,A -85,B 0,C 180,E1 -15639.515,E2 -15639.515} C_VEL
LIN {X 0,Y 316.875,Z 424.614,A -85,B 0,C 180,E1 -15639.96,E2 -15639.96} C_VEL
LIN {X 0,Y 320.251,Z 435.128,A -85,B 0,C 180,E1 -15641.776,E2 -15641.776} C_VEL
LIN {X 0,Y 321.955,Z 443.609,A -85,B 0,C 180,E1 -15643.273,E2 -15643.273} C_VEL
LIN {X 0,Y 322.474,Z 449.281,A -85,B 0,C 180,E1 -15644.29,E2 -15644.29} C_VEL
LIN {X 0,Y 320.723,Z 457.703,A -85,B 0,C 180,E1 -15645.728,E2 -15645.728} C_VEL
LIN {X 0,Y 318.872,Z 464.886,A -85,B 0,C 180,E1 -15647.267,E2 -15647.267} C_VEL
LIN {X 0,Y 317.278,Z 470.611,A -85,B 0,C 180,E1 -15648.824,E2 -15648.824} C_VEL
LIN {X 0,Y 315.849,Z 475.052,A -85,B 0,C 180,E1 -15650.393,E2 -15650.393} C_VEL
LIN {X 0,Y 314.335,Z 478.898,A -85,B 0,C 180,E1 -15652.291,E2 -15652.291} C_VEL
LIN {X 0,Y 313.506,Z 480.624,A -85,B 0,C 180,E1 -15653.564,E2 -15653.564} C_VEL
LIN {X 0,Y 312.799,Z 481.741,A -85,B 0,C 180,E1 -15654.844,E2 -15654.844} C_VEL
LIN {X 0,Y 312.194,Z 482.234,A -85,B 0,C 180,E1 -15656.128,E2 -15656.128} C_VEL
LIN {X 0,Y 311.818,Z 482.087,A -85,B 0,C 180,E1 -15657.416,E2 -15657.416} C_VEL
LIN {X 0,Y 311.591,Z 481.293,A -85,B 0,C 180,E1 -15658.708,E2 -15658.708} C_VEL
LIN {X 0,Y 311.374,Z 478.91,A -85,B 0,C 180,E1 -15660.647,E2 -15660.647} C_VEL
LIN {X 0,Y 311.417,Z 475,A -85,B 0,C 180,E1 -15662.587,E2 -15662.587} C_VEL
LIN {X 0,Y 311.705,Z 469.391,A -85,B 0,C 180,E1 -15664.526,E2 -15664.526} C_VEL
LIN {X 0,Y 312.018,Z 463.194,A -85,B 0,C 180,E1 -15666.142,E2 -15666.142} C_VEL
LIN {X 0,Y 312.271,Z 455.282,A -85,B 0,C 180,E1 -15667.761,E2 -15667.761} C_VEL
LIN {X 0,Y 312.636,Z 446.221,A -85,B 0,C 180,E1 -15669.217,E2 -15669.217} C_VEL
LIN {X 0,Y 313.167,Z 435.926,A -85,B 0,C 180,E1 -15670.506,E2 -15670.506} C_VEL
LIN {X 0,Y 313.42,Z 431.275,A -85,B 0,C 180,E1 -15670.988,E2 -15670.988} C_VEL
LIN {X 0,Y 312.138,Z 420.464,A -85,B 0,C 180,E1 -15671.939,E2 -15671.939} C_VEL
LIN {X 0,Y 311.419,Z 412.781,A -85,B 0,C 180,E1 -15672.463,E2 -15672.463} C_VEL
LIN {X 0,Y 311.607,Z 406.213,A -85,B 0,C 180,E1 -15676.375,E2 -15676.375} C_VEL
LIN {X 0,Y 311.954,Z 399.531,A -85,B 0,C 180,E1 -15680.439,E2 -15680.439} C_VEL
LIN {X 0,Y 312.297,Z 392.851,A -85,B 0,C 180,E1 -15684.603,E2 -15684.603} C_VEL
LIN {X 0,Y 312.761,Z 386.257,A -85,B 0,C 180,E1 -15688.793,E2 -15688.793} C_VEL
LIN {X 0,Y 312.826,Z 381.971,A -85,B 0,C 180,E1 -15691.587,E2 -15691.587} C_VEL
LIN {X 0,Y 312.697,Z 381.534,A -85,B 0,C 180,E1 -15691.969,E2 -15691.969} C_VEL
LIN {X 0,Y 312.541,Z 381.55,A -85,B 0,C 180,E1 -15695.95,E2 -15695.95} C_VEL
LIN {X 0,Y 312.506,Z 381.555,A -85,B 0,C 180,E1 -15700.125,E2 -15700.125} C_VEL
LIN {X 0,Y 312.483,Z 381.558,A -85,B 0,C 180,E1 -15703.969,E2 -15703.969} C_VEL
LIN {X 0,Y 312.489,Z 381.557,A -85,B 0,C 180,E1 -15707.918,E2 -15707.918} C_VEL
LIN {X 0,Y 312.501,Z 381.558,A -85,B 0,C 180,E1 -15710.971,E2 -15710.971} C_VEL
LIN {X 0,Y 312.535,Z 381.553,A -85,B 0,C 180,E1 -15714.22,E2 -15714.22} C_VEL
LIN {X 0,Y 312.506,Z 381.555,A -85,B 0,C 180,E1 -15717.334,E2 -15717.334} C_VEL
LIN {X 0,Y 312.547,Z 381.55,A -85,B 0,C 180,E1 -15721.279,E2 -15721.279} C_VEL
LIN {X 0,Y 312.588,Z 381.547,A -85,B 0,C 180,E1 -15724.711,E2 -15724.711} C_VEL
LIN {X 0,Y 312.59,Z 381.544,A -85,B 0,C 180,E1 -15727.529,E2 -15727.529} C_VEL
LIN {X 0,Y 312.642,Z 381.539,A -85,B 0,C 180,E1 -15731.656,E2 -15731.656} C_VEL
LIN {X 0,Y 312.697,Z 381.532,A -85,B 0,C 180,E1 -15735.686,E2 -15735.686} C_VEL
LIN {X 0,Y 312.702,Z 381.532,A -85,B 0,C 180,E1 -15739.642,E2 -15739.642} C_VEL
LIN {X 0,Y 312.857,Z 381.516,A -85,B 0,C 180,E1 -15742.254,E2 -15742.254} C_VEL
LIN {X 0,Y 312.718,Z 381.528,A -85,B 0,C 180,E1 -15744.842,E2 -15744.842} C_VEL
LIN {X 0,Y 312.992,Z 381.495,A -85,B 0,C 180,E1 -15748.713,E2 -15748.713} C_VEL
LIN {X 0,Y 312.994,Z 381.495,A -85,B 0,C 180,E1 -15751.287,E2 -15751.287} C_VEL
LIN {X 0,Y 312.719,Z 381.528,A -85,B 0,C 180,E1 -15755.158,E2 -15755.158} C_VEL
LIN {X 0,Y 312.869,Z 381.514,A -85,B 0,C 180,E1 -15757.746,E2 -15757.746} C_VEL
LIN {X 0,Y 312.673,Z 381.538,A -85,B 0,C 180,E1 -15761.671,E2 -15761.671} C_VEL
LIN {X 0,Y 312.703,Z 381.53,A -85,B 0,C 180,E1 -15764.888,E2 -15764.888} C_VEL
LIN {X 0,Y 312.636,Z 381.54,A -85,B 0,C 180,E1 -15769.238,E2 -15769.238} C_VEL
LIN {X 0,Y 312.549,Z 381.549,A -85,B 0,C 180,E1 -15772.789,E2 -15772.789} C_VEL
LIN {X 0,Y 312.605,Z 381.545,A -85,B 0,C 180,E1 -15775.935,E2 -15775.935} C_VEL
LIN {X 0,Y 312.54,Z 381.554,A -85,B 0,C 180,E1 -15779.65,E2 -15779.65} C_VEL
LIN {X 0,Y 312.521,Z 381.556,A -85,B 0,C 180,E1 -15783.689,E2 -15783.689} C_VEL
LIN {X 0,Y 312.54,Z 381.556,A -85,B 0,C 180,E1 -15787.383,E2 -15787.383} C_VEL
LIN {X 0,Y 312.492,Z 381.557,A -85,B 0,C 180,E1 -15790.709,E2 -15790.709} C_VEL
LIN {X 0,Y 312.453,Z 381.561,A -85,B 0,C 180,E1 -15794.209,E2 -15794.209} C_VEL
LIN {X 0,Y 312.486,Z 381.558,A -85,B 0,C 180,E1 -15797.918,E2 -15797.918} C_VEL
LIN {X 0,Y 312.5,Z 381.559,A -85,B 0,C 180,E1 -15800.971,E2 -15800.971} C_VEL
LIN {X 0,Y 312.534,Z 381.551,A -85,B 0,C 180,E1 -15804.22,E2 -15804.22} C_VEL
LIN {X 0,Y 312.506,Z 381.558,A -85,B 0,C 180,E1 -15807.334,E2 -15807.334} C_VEL
LIN {X 0,Y 312.554,Z 381.552,A -85,B 0,C 180,E1 -15811.276,E2 -15811.276} C_VEL
LIN {X 0,Y 312.587,Z 381.548,A -85,B 0,C 180,E1 -15814.711,E2 -15814.711} C_VEL
LIN {X 0,Y 312.589,Z 381.545,A -85,B 0,C 180,E1 -15817.529,E2 -15817.529} C_VEL
LIN {X 0,Y 312.64,Z 381.538,A -85,B 0,C 180,E1 -15821.656,E2 -15821.656} C_VEL
LIN {X 0,Y 312.696,Z 381.531,A -85,B 0,C 180,E1 -15825.686,E2 -15825.686} C_VEL
LIN {X 0,Y 312.71,Z 381.528,A -85,B 0,C 180,E1 -15829.91,E2 -15829.91} C_VEL
LIN {X 0,Y 312.912,Z 381.504,A -85,B 0,C 180,E1 -15833.552,E2 -15833.552} C_VEL
LIN {X 0,Y 312.687,Z 381.532,A -85,B 0,C 180,E1 -15835.505,E2 -15835.505} C_VEL
LIN {X 0,Y 312.048,Z 381.617,A -85,B 0,C 180,E1 -15836.582,E2 -15836.582} C_VEL
LIN {X 0,Y 309.335,Z 381.953,A -85,B 0,C 180,E1 -15838.339,E2 -15838.339} C_VEL
LIN {X 0,Y 307.036,Z 382.236,A -85,B 0,C 180,E1 -15839.764,E2 -15839.764} C_VEL
LIN {X 0,Y 306.046,Z 382.362,A -85,B 0,C 180,E1 -15840.864,E2 -15840.864} C_VEL
LIN {X 0,Y 305.963,Z 382.369,A -85,B 0,C 180,E1 -15841.236,E2 -15841.236} C_VEL
LIN {X 0,Y 305.65,Z 382.41,A -85,B 0,C 180,E1 -15843.955,E2 -15843.955} C_VEL
LIN {X 0,Y 305.855,Z 382.387,A -85,B 0,C 180,E1 -15846.597,E2 -15846.597} C_VEL
LIN {X 0,Y 305.737,Z 382.398,A -85,B 0,C 180,E1 -15849.26,E2 -15849.26} C_VEL
LIN {X 0,Y 305.59,Z 382.416,A -85,B 0,C 180,E1 -15853.296,E2 -15853.296} C_VEL
LIN {X 0,Y 305.595,Z 382.419,A -85,B 0,C 180,E1 -15856.02,E2 -15856.02} C_VEL
LIN {X 0,Y 305.578,Z 382.418,A -85,B 0,C 180,E1 -15859.445,E2 -15859.445} C_VEL
LIN {X 0,Y 305.492,Z 382.429,A -85,B 0,C 180,E1 -15863.041,E2 -15863.041} C_VEL
LIN {X 0,Y 305.548,Z 382.425,A -85,B 0,C 180,E1 -15866.227,E2 -15866.227} C_VEL
LIN {X 0,Y 305.489,Z 382.429,A -85,B 0,C 180,E1 -15869.047,E2 -15869.047} C_VEL
LIN {X 0,Y 305.444,Z 382.44,A -85,B 0,C 180,E1 -15871.952,E2 -15871.952} C_VEL
LIN {X 0,Y 305.464,Z 382.432,A -85,B 0,C 180,E1 -15875.113,E2 -15875.113} C_VEL
LIN {X 0,Y 305.469,Z 382.432,A -85,B 0,C 180,E1 -15878.533,E2 -15878.533} C_VEL
LIN {X 0,Y 305.461,Z 382.432,A -85,B 0,C 180,E1 -15882.587,E2 -15882.587} C_VEL
LIN {X 0,Y 305.474,Z 382.432,A -85,B 0,C 180,E1 -15886.354,E2 -15886.354} C_VEL
LIN {X 0,Y 305.487,Z 382.438,A -85,B 0,C 180,E1 -15889.393,E2 -15889.393} C_VEL
LIN {X 0,Y 307.265,Z 391.443,A -85,B 0,C 180,E1 -15893.182,E2 -15893.182} C_VEL
LIN {X 0,Y 309.364,Z 401.438,A -85,B 0,C 180,E1 -15897.198,E2 -15897.198} C_VEL
LIN {X 0,Y 310.43,Z 406.976,A -85,B 0,C 180,E1 -15899.351,E2 -15899.351} C_VEL
LIN {X 0,Y 308.853,Z 415.889,A -85,B 0,C 180,E1 -15902.555,E2 -15902.555} C_VEL
LIN {X 0,Y 306.805,Z 428.528,A -85,B 0,C 180,E1 -15907.082,E2 -15907.082} C_VEL
LIN {X 0,Y 305.55,Z 439.53,A -85,B 0,C 180,E1 -15911.015,E2 -15911.015} C_VEL
LIN {X 0,Y 306.063,Z 452.653,A -85,B 0,C 180,E1 -15911.638,E2 -15911.638} C_VEL
LIN {X 0,Y 306.902,Z 465.325,A -85,B 0,C 180,E1 -15912.509,E2 -15912.509} C_VEL
LIN {X 0,Y 307.346,Z 473.485,A -85,B 0,C 180,E1 -15913.22,E2 -15913.22} C_VEL
LIN {X 0,Y 306.619,Z 485.202,A -85,B 0,C 180,E1 -15914.496,E2 -15914.496} C_VEL
LIN {X 0,Y 305.818,Z 495.198,A -85,B 0,C 180,E1 -15915.867,E2 -15915.867} C_VEL
LIN {X 0,Y 305.275,Z 504.021,A -85,B 0,C 180,E1 -15917.367,E2 -15917.367} C_VEL
LIN {X 0,Y 304.789,Z 512.042,A -85,B 0,C 180,E1 -15919.034,E2 -15919.034} C_VEL
LIN {X 0,Y 304.492,Z 519.778,A -85,B 0,C 180,E1 -15921.037,E2 -15921.037} C_VEL
LIN {X 0,Y 304.427,Z 525.911,A -85,B 0,C 180,E1 -15923.072,E2 -15923.072} C_VEL
LIN {X 0,Y 304.451,Z 529.777,A -85,B 0,C 180,E1 -15924.702,E2 -15924.702} C_VEL
LIN {X 0,Y 304.445,Z 532.304,A -85,B 0,C 180,E1 -15926.029,E2 -15926.029} C_VEL
LIN {X 0,Y 304.572,Z 534.299,A -85,B 0,C 180,E1 -15927.355,E2 -15927.355} C_VEL
LIN {X 0,Y 304.506,Z 535.773,A -85,B 0,C 180,E1 -15928.678,E2 -15928.678} C_VEL
LIN {X 0,Y 304.444,Z 536.801,A -85,B 0,C 180,E1 -15930,E2 -15930} C_VEL
LIN {X 0,Y 304.457,Z 537.341,A -85,B 0,C 180,E1 -15931.323,E2 -15931.323} C_VEL
LIN {X 0,Y 304.267,Z 537.437,A -85,B 0,C 180,E1 -15932.648,E2 -15932.648} C_VEL
LIN {X 0,Y 304.041,Z 537.107,A -85,B 0,C 180,E1 -15933.977,E2 -15933.977} C_VEL
LIN {X 0,Y 303.96,Z 535.622,A -85,B 0,C 180,E1 -15936.16,E2 -15936.16} C_VEL
LIN {X 0,Y 304.039,Z 532.557,A -85,B 0,C 180,E1 -15938.642,E2 -15938.642} C_VEL
LIN {X 0,Y 304.439,Z 528.985,A -85,B 0,C 180,E1 -15940.643,E2 -15940.643} C_VEL
LIN {X 0,Y 305.261,Z 524.36,A -85,B 0,C 180,E1 -15942.634,E2 -15942.634} C_VEL
LIN {X 0,Y 306.699,Z 517.453,A -85,B 0,C 180,E1 -15944.939,E2 -15944.939} C_VEL
LIN {X 0,Y 308.427,Z 509.833,A -85,B 0,C 180,E1 -15946.948,E2 -15946.948} C_VEL
LIN {X 0,Y 310.547,Z 500.946,A -85,B 0,C 180,E1 -15948.814,E2 -15948.814} C_VEL
LIN {X 0,Y 312.961,Z 490.685,A -85,B 0,C 180,E1 -15950.542,E2 -15950.542} C_VEL
LIN {X 0,Y 314.999,Z 480.364,A -85,B 0,C 180,E1 -15951.945,E2 -15951.945} C_VEL
LIN {X 0,Y 316.001,Z 469.646,A -85,B 0,C 180,E1 -15953.243,E2 -15953.243} C_VEL
LIN {X 0,Y 315.606,Z 459.59,A -85,B 0,C 180,E1 -15954.404,E2 -15954.404} C_VEL
LIN {X 0,Y 313.834,Z 447.113,A -85,B 0,C 180,E1 -15955.788,E2 -15955.788} C_VEL
LIN {X 0,Y 311.283,Z 436.113,A -85,B 0,C 180,E1 -15957.025,E2 -15957.025} C_VEL
LIN {X 0,Y 314.42,Z 427.242,A -85,B 0,C 180,E1 -15960.938,E2 -15960.938} C_VEL
LIN {X 0,Y 315.28,Z 424.414,A -85,B 0,C 180,E1 -15962.344,E2 -15962.344} C_VEL
LIN {X 0,Y 314.988,Z 421.239,A -85,B 0,C 180,E1 -15964.356,E2 -15964.356} C_VEL
LIN {X 0,Y 314.158,Z 417.648,A -85,B 0,C 180,E1 -15967.158,E2 -15967.158} C_VEL
LIN {X 0,Y 313.45,Z 414.192,A -85,B 0,C 180,E1 -15970.559,E2 -15970.559} C_VEL
LIN {X 0,Y 312.831,Z 411.719,A -85,B 0,C 180,E1 -15974.142,E2 -15974.142} C_VEL
LIN {X 0,Y 312.589,Z 410.878,A -85,B 0,C 180,E1 -15976.01,E2 -15976.01} C_VEL
LIN {X 0,Y 312.118,Z 410.106,A -85,B 0,C 180,E1 -15979.959,E2 -15979.959} C_VEL
LIN {X 0,Y 311.954,Z 410.236,A -85,B 0,C 180,E1 -15982.535,E2 -15982.535} C_VEL
LIN {X 0,Y 311.704,Z 411.1,A -85,B 0,C 180,E1 -15985.69,E2 -15985.69} C_VEL
LIN {X 0,Y 311.557,Z 411.754,A -85,B 0,C 180,E1 -15987.222,E2 -15987.222} C_VEL
LIN {X 0,Y 310.872,Z 413.59,A -85,B 0,C 180,E1 -15990.174,E2 -15990.174} C_VEL
LIN {X 0,Y 309.94,Z 415.884,A -85,B 0,C 180,E1 -15993.031,E2 -15993.031} C_VEL
LIN {X 0,Y 308.699,Z 419.855,A -85,B 0,C 180,E1 -15997.23,E2 -15997.23} C_VEL
LIN {X 0,Y 308.557,Z 420.821,A -85,B 0,C 180,E1 -15997.995,E2 -15997.995} C_VEL
LIN {X 0,Y 309.628,Z 423.729,A -85,B 0,C 180,E1 -15998.534,E2 -15998.534} C_VEL
LIN {X 0,Y 311.841,Z 429.333,A -85,B 0,C 180,E1 -15999.623,E2 -15999.623} C_VEL
LIN {X 0,Y 314.147,Z 437.086,A -85,B 0,C 180,E1 -16001.071,E2 -16001.071} C_VEL
LIN {X 0,Y 315.877,Z 446.058,A -85,B 0,C 180,E1 -16002.759,E2 -16002.759} C_VEL
LIN {X 0,Y 316.176,Z 452.317,A -85,B 0,C 180,E1 -16003.969,E2 -16003.969} C_VEL
LIN {X 0,Y 314.181,Z 460.294,A -85,B 0,C 180,E1 -16005.425,E2 -16005.425} C_VEL
LIN {X 0,Y 312.216,Z 467.131,A -85,B 0,C 180,E1 -16006.991,E2 -16006.991} C_VEL
LIN {X 0,Y 310.207,Z 473.401,A -85,B 0,C 180,E1 -16008.897,E2 -16008.897} C_VEL
LIN {X 0,Y 308.488,Z 477.998,A -85,B 0,C 180,E1 -16010.824,E2 -16010.824} C_VEL
LIN {X 0,Y 307.436,Z 480.237,A -85,B 0,C 180,E1 -16012.117,E2 -16012.117} C_VEL
LIN {X 0,Y 306.549,Z 481.81,A -85,B 0,C 180,E1 -16013.418,E2 -16013.418} C_VEL
LIN {X 0,Y 305.8,Z 482.746,A -85,B 0,C 180,E1 -16014.725,E2 -16014.725} C_VEL
LIN {X 0,Y 305.17,Z 483.068,A -85,B 0,C 180,E1 -16016.038,E2 -16016.038} C_VEL
LIN {X 0,Y 304.784,Z 482.771,A -85,B 0,C 180,E1 -16017.357,E2 -16017.357} C_VEL
LIN {X 0,Y 304.518,Z 481.845,A -85,B 0,C 180,E1 -16018.678,E2 -16018.678} C_VEL
LIN {X 0,Y 304.3,Z 479.254,A -85,B 0,C 180,E1 -16020.662,E2 -16020.662} C_VEL
LIN {X 0,Y 304.325,Z 475.139,A -85,B 0,C 180,E1 -16022.647,E2 -16022.647} C_VEL
LIN {X 0,Y 304.622,Z 469.307,A -85,B 0,C 180,E1 -16024.632,E2 -16024.632} C_VEL
LIN {X 0,Y 304.948,Z 462.882,A -85,B 0,C 180,E1 -16026.285,E2 -16026.285} C_VEL
LIN {X 0,Y 305.221,Z 454.661,A -85,B 0,C 180,E1 -16027.941,E2 -16027.941} C_VEL
LIN {X 0,Y 305.609,Z 445.24,A -85,B 0,C 180,E1 -16029.431,E2 -16029.431} C_VEL
LIN {X 0,Y 306.196,Z 434.542,A -85,B 0,C 180,E1 -16030.748,E2 -16030.748} C_VEL
LIN {X 0,Y 306.059,Z 429.55,A -85,B 0,C 180,E1 -16031.256,E2 -16031.256} C_VEL
LIN {X 0,Y 304.782,Z 418.005,A -85,B 0,C 180,E1 -16032.231,E2 -16032.231} C_VEL
LIN {X 0,Y 304.353,Z 413.062,A -85,B 0,C 180,E1 -16032.587,E2 -16032.587} C_VEL
LIN {X 0,Y 304.563,Z 406.163,A -85,B 0,C 180,E1 -16036.765,E2 -16036.765} C_VEL
LIN {X 0,Y 304.887,Z 400.553,A -85,B 0,C 180,E1 -16040.229,E2 -16040.229} C_VEL
LIN {X 0,Y 305.225,Z 393.818,A -85,B 0,C 180,E1 -16044.486,E2 -16044.486} C_VEL
LIN {X 0,Y 305.772,Z 386.591,A -85,B 0,C 180,E1 -16049.142,E2 -16049.142} C_VEL
LIN {X 0,Y 305.756,Z 382.706,A -85,B 0,C 180,E1 -16051.737,E2 -16051.737} C_VEL
LIN {X 0,Y 305.608,Z 382.417,A -85,B 0,C 180,E1 -16052.322,E2 -16052.322} C_VEL
LIN {X 0,Y 305.476,Z 382.434,A -85,B 0,C 180,E1 -16056.74,E2 -16056.74} C_VEL
LIN {X 0,Y 305.457,Z 382.436,A -85,B 0,C 180,E1 -16060.6,E2 -16060.6} C_VEL
LIN {X 0,Y 305.421,Z 382.44,A -85,B 0,C 180,E1 -16064.493,E2 -16064.493} C_VEL
LIN {X 0,Y 305.445,Z 382.436,A -85,B 0,C 180,E1 -16068.143,E2 -16068.143} C_VEL
LIN {X 0,Y 305.47,Z 382.431,A -85,B 0,C 180,E1 -16071.596,E2 -16071.596} C_VEL
LIN {X 0,Y 305.465,Z 382.435,A -85,B 0,C 180,E1 -16074.887,E2 -16074.887} C_VEL
LIN {X 0,Y 305.452,Z 382.437,A -85,B 0,C 180,E1 -16078.356,E2 -16078.356} C_VEL
LIN {X 0,Y 305.516,Z 382.426,A -85,B 0,C 180,E1 -16081.113,E2 -16081.113} C_VEL
LIN {X 0,Y 305.574,Z 382.421,A -85,B 0,C 180,E1 -16084.088,E2 -16084.088} C_VEL
LIN {X 0,Y 305.529,Z 382.429,A -85,B 0,C 180,E1 -16088.405,E2 -16088.405} C_VEL
LIN {X 0,Y 305.594,Z 382.416,A -85,B 0,C 180,E1 -16091.218,E2 -16091.218} C_VEL
LIN {X 0,Y 305.652,Z 382.409,A -85,B 0,C 180,E1 -16095.349,E2 -16095.349} C_VEL
LIN {X 0,Y 305.639,Z 382.41,A -85,B 0,C 180,E1 -16099.4,E2 -16099.4} C_VEL
LIN {X 0,Y 305.8,Z 382.395,A -85,B 0,C 180,E1 -16102.074,E2 -16102.074} C_VEL
LIN {X 0,Y 305.689,Z 382.404,A -85,B 0,C 180,E1 -16104.723,E2 -16104.723} C_VEL
LIN {X 0,Y 305.959,Z 382.371,A -85,B 0,C 180,E1 -16108.684,E2 -16108.684} C_VEL
LIN {X 0,Y 305.961,Z 382.371,A -85,B 0,C 180,E1 -16111.316,E2 -16111.316} C_VEL
LIN {X 0,Y 305.849,Z 382.384,A -85,B 0,C 180,E1 -16116.597,E2 -16116.597} C_VEL
LIN {X 0,Y 305.739,Z 382.399,A -85,B 0,C 180,E1 -16119.26,E2 -16119.26} C_VEL
LIN {X 0,Y 305.592,Z 382.417,A -85,B 0,C 180,E1 -16123.296,E2 -16123.296} C_VEL
LIN {X 0,Y 305.597,Z 382.418,A -85,B 0,C 180,E1 -16126.02,E2 -16126.02} C_VEL
LIN {X 0,Y 305.584,Z 382.42,A -85,B 0,C 180,E1 -16129.447,E2 -16129.447} C_VEL
LIN {X 0,Y 305.494,Z 382.429,A -85,B 0,C 180,E1 -16133.042,E2 -16133.042} C_VEL
LIN {X 0,Y 305.534,Z 382.424,A -85,B 0,C 180,E1 -16136.221,E2 -16136.221} C_VEL
LIN {X 0,Y 305.49,Z 382.43,A -85,B 0,C 180,E1 -16139.047,E2 -16139.047} C_VEL
LIN {X 0,Y 305.444,Z 382.436,A -85,B 0,C 180,E1 -16141.952,E2 -16141.952} C_VEL
LIN {X 0,Y 305.465,Z 382.435,A -85,B 0,C 180,E1 -16145.113,E2 -16145.113} C_VEL
LIN {X 0,Y 305.469,Z 382.431,A -85,B 0,C 180,E1 -16148.533,E2 -16148.533} C_VEL
LIN {X 0,Y 305.457,Z 382.434,A -85,B 0,C 180,E1 -16152.586,E2 -16152.586} C_VEL
LIN {X 0,Y 305.427,Z 382.436,A -85,B 0,C 180,E1 -16156.345,E2 -16156.345} C_VEL
LIN {X 0,Y 305.459,Z 382.433,A -85,B 0,C 180,E1 -16159.892,E2 -16159.892} C_VEL
LIN {X 0,Y 305.482,Z 382.431,A -85,B 0,C 180,E1 -16163.632,E2 -16163.632} C_VEL
LIN {X 0,Y 305.467,Z 382.432,A -85,B 0,C 180,E1 -16166.483,E2 -16166.483} C_VEL
LIN {X 0,Y 305.498,Z 382.433,A -85,B 0,C 180,E1 -16170.95,E2 -16170.95} C_VEL
LIN {X 0,Y 305.573,Z 382.418,A -85,B 0,C 180,E1 -16174.088,E2 -16174.088} C_VEL
LIN {X 0,Y 305.503,Z 382.429,A -85,B 0,C 180,E1 -16178.403,E2 -16178.403} C_VEL
LIN {X 0,Y 305.592,Z 382.418,A -85,B 0,C 180,E1 -16181.218,E2 -16181.218} C_VEL
LIN {X 0,Y 305.651,Z 382.41,A -85,B 0,C 180,E1 -16185.349,E2 -16185.349} C_VEL
LIN {X 0,Y 305.643,Z 382.41,A -85,B 0,C 180,E1 -16189.4,E2 -16189.4} C_VEL
LIN {X 0,Y 305.815,Z 382.389,A -85,B 0,C 180,E1 -16192.074,E2 -16192.074} C_VEL
LIN {X 0,Y 305.691,Z 382.408,A -85,B 0,C 180,E1 -16194.723,E2 -16194.723} C_VEL
LIN {X 0,Y 305.959,Z 382.374,A -85,B 0,C 180,E1 -16198.684,E2 -16198.684} C_VEL
LIN {X 0,Y 305.963,Z 382.369,A -85,B 0,C 180,E1 -16201.236,E2 -16201.236} C_VEL
LIN {X 0,Y 305.285,Z 382.459,A -85,B 0,C 180,E1 -16202.331,E2 -16202.331} C_VEL
LIN {X 0,Y 302.413,Z 382.82,A -85,B 0,C 180,E1 -16204.114,E2 -16204.114} C_VEL
LIN {X 0,Y 299.961,Z 383.123,A -85,B 0,C 180,E1 -16205.559,E2 -16205.559} C_VEL
LIN {X 0,Y 298.88,Z 383.255,A -85,B 0,C 180,E1 -16206.679,E2 -16206.679} C_VEL
LIN {X 0,Y 298.776,Z 383.265,A -85,B 0,C 180,E1 -16207.059,E2 -16207.059} C_VEL
LIN {X 0,Y 298.682,Z 383.276,A -85,B 0,C 180,E1 -16209.48,E2 -16209.48} C_VEL
LIN {X 0,Y 298.554,Z 383.294,A -85,B 0,C 180,E1 -16213.615,E2 -16213.615} C_VEL
LIN {X 0,Y 298.55,Z 383.296,A -85,B 0,C 180,E1 -16216.409,E2 -16216.409} C_VEL
LIN {X 0,Y 298.513,Z 383.299,A -85,B 0,C 180,E1 -16219.655,E2 -16219.655} C_VEL
LIN {X 0,Y 298.459,Z 383.306,A -85,B 0,C 180,E1 -16223.598,E2 -16223.598} C_VEL
LIN {X 0,Y 298.49,Z 383.302,A -85,B 0,C 180,E1 -16226.574,E2 -16226.574} C_VEL
LIN {X 0,Y 298.418,Z 383.312,A -85,B 0,C 180,E1 -16229.641,E2 -16229.641} C_VEL
LIN {X 0,Y 298.396,Z 383.312,A -85,B 0,C 180,E1 -16232.8,E2 -16232.8} C_VEL
LIN {X 0,Y 298.466,Z 383.304,A -85,B 0,C 180,E1 -16236.812,E2 -16236.812} C_VEL
LIN {X 0,Y 298.39,Z 383.314,A -85,B 0,C 180,E1 -16241.088,E2 -16241.088} C_VEL
LIN {X 0,Y 298.389,Z 383.313,A -85,B 0,C 180,E1 -16245.041,E2 -16245.041} C_VEL
LIN {X 0,Y 298.429,Z 383.308,A -85,B 0,C 180,E1 -16248.903,E2 -16248.903} C_VEL
LIN {X 0,Y 298.498,Z 383.563,A -85,B 0,C 180,E1 -16249.173,E2 -16249.173} C_VEL
LIN {X 0,Y 300.147,Z 391.838,A -85,B 0,C 180,E1 -16252.761,E2 -16252.761} C_VEL
LIN {X 0,Y 302.412,Z 402.797,A -85,B 0,C 180,E1 -16257.283,E2 -16257.283} C_VEL
LIN {X 0,Y 303.377,Z 408.04,A -85,B 0,C 180,E1 -16259.36,E2 -16259.36} C_VEL
LIN {X 0,Y 301.539,Z 417.785,A -85,B 0,C 180,E1 -16262.968,E2 -16262.968} C_VEL
LIN {X 0,Y 299.636,Z 429.353,A -85,B 0,C 180,E1 -16267.231,E2 -16267.231} C_VEL
LIN {X 0,Y 298.477,Z 439.267,A -85,B 0,C 180,E1 -16270.887,E2 -16270.887} C_VEL
LIN {X 0,Y 298.911,Z 451.747,A -85,B 0,C 180,E1 -16271.494,E2 -16271.494} C_VEL
LIN {X 0,Y 299.681,Z 463.968,A -85,B 0,C 180,E1 -16272.338,E2 -16272.338} C_VEL
LIN {X 0,Y 300.257,Z 473.217,A -85,B 0,C 180,E1 -16273.163,E2 -16273.163} C_VEL
LIN {X 0,Y 299.571,Z 484.483,A -85,B 0,C 180,E1 -16274.423,E2 -16274.423} C_VEL
LIN {X 0,Y 298.753,Z 494.775,A -85,B 0,C 180,E1 -16275.873,E2 -16275.873} C_VEL
LIN {X 0,Y 298.209,Z 503.547,A -85,B 0,C 180,E1 -16277.409,E2 -16277.409} C_VEL
LIN {X 0,Y 297.734,Z 511.523,A -85,B 0,C 180,E1 -16279.115,E2 -16279.115} C_VEL
LIN {X 0,Y 297.438,Z 519.213,A -85,B 0,C 180,E1 -16281.165,E2 -16281.165} C_VEL
LIN {X 0,Y 297.391,Z 525.225,A -85,B 0,C 180,E1 -16283.214,E2 -16283.214} C_VEL
LIN {X 0,Y 297.406,Z 529.822,A -85,B 0,C 180,E1 -16285.256,E2 -16285.256} C_VEL
LIN {X 0,Y 297.531,Z 533.174,A -85,B 0,C 180,E1 -16287.292,E2 -16287.292} C_VEL
LIN {X 0,Y 297.476,Z 534.724,A -85,B 0,C 180,E1 -16288.646,E2 -16288.646} C_VEL
LIN {X 0,Y 297.411,Z 535.82,A -85,B 0,C 180,E1 -16290,E2 -16290} C_VEL
LIN {X 0,Y 297.41,Z 536.481,A -85,B 0,C 180,E1 -16291.354,E2 -16291.354} C_VEL
LIN {X 0,Y 297.2,Z 536.635,A -85,B 0,C 180,E1 -16292.711,E2 -16292.711} C_VEL
LIN {X 0,Y 296.906,Z 535.716,A -85,B 0,C 180,E1 -16295.433,E2 -16295.433} C_VEL
LIN {X 0,Y 296.938,Z 533.079,A -85,B 0,C 180,E1 -16298.164,E2 -16298.164} C_VEL
LIN {X 0,Y 297.234,Z 529.99,A -85,B 0,C 180,E1 -16300.215,E2 -16300.215} C_VEL
LIN {X 0,Y 297.911,Z 525.9,A -85,B 0,C 180,E1 -16302.258,E2 -16302.258} C_VEL
LIN {X 0,Y 299.373,Z 519.713,A -85,B 0,C 180,E1 -16304.618,E2 -16304.618} C_VEL
LIN {X 0,Y 300.835,Z 513.475,A -85,B 0,C 180,E1 -16306.509,E2 -16306.509} C_VEL
LIN {X 0,Y 303.079,Z 504.907,A -85,B 0,C 180,E1 -16308.593,E2 -16308.593} C_VEL
LIN {X 0,Y 305.672,Z 494.822,A -85,B 0,C 180,E1 -16310.526,E2 -16310.526} C_VEL
LIN {X 0,Y 308.2,Z 484.464,A -85,B 0,C 180,E1 -16312.102,E2 -16312.102} C_VEL
LIN {X 0,Y 309.779,Z 473.053,A -85,B 0,C 180,E1 -16313.612,E2 -16313.612} C_VEL
LIN {X 0,Y 309.797,Z 463.128,A -85,B 0,C 180,E1 -16314.847,E2 -16314.847} C_VEL
LIN {X 0,Y 308.574,Z 451.418,A -85,B 0,C 180,E1 -16316.261,E2 -16316.261} C_VEL
LIN {X 0,Y 305.833,Z 438.719,A -85,B 0,C 180,E1 -16317.826,E2 -16317.826} C_VEL
LIN {X 0,Y 305.214,Z 435.584,A -85,B 0,C 180,E1 -16318.214,E2 -16318.214} C_VEL
LIN {X 0,Y 308.091,Z 428.157,A -85,B 0,C 180,E1 -16321.646,E2 -16321.646} C_VEL
LIN {X 0,Y 308.559,Z 426.431,A -85,B 0,C 180,E1 -16322.569,E2 -16322.569} C_VEL
LIN {X 0,Y 308.179,Z 423.085,A -85,B 0,C 180,E1 -16324.817,E2 -16324.817} C_VEL
LIN {X 0,Y 307.273,Z 419.081,A -85,B 0,C 180,E1 -16328.138,E2 -16328.138} C_VEL
LIN {X 0,Y 306.772,Z 416.503,A -85,B 0,C 180,E1 -16330.886,E2 -16330.886} C_VEL
LIN {X 0,Y 306.293,Z 414.672,A -85,B 0,C 180,E1 -16333.501,E2 -16333.501} C_VEL
LIN {X 0,Y 305.895,Z 413.336,A -85,B 0,C 180,E1 -16336.429,E2 -16336.429} C_VEL
LIN {X 0,Y 305.491,Z 412.655,A -85,B 0,C 180,E1 -16339.897,E2 -16339.897} C_VEL
LIN {X 0,Y 305.202,Z 412.93,A -85,B 0,C 180,E1 -16343.703,E2 -16343.703} C_VEL
LIN {X 0,Y 304.964,Z 413.778,A -85,B 0,C 180,E1 -16346.421,E2 -16346.421} C_VEL
LIN {X 0,Y 304.306,Z 415.405,A -85,B 0,C 180,E1 -16349.463,E2 -16349.463} C_VEL
LIN {X 0,Y 303.355,Z 417.55,A -85,B 0,C 180,E1 -16352.396,E2 -16352.396} C_VEL
LIN {X 0,Y 302.033,Z 421.325,A -85,B 0,C 180,E1 -16356.608,E2 -16356.608} C_VEL
LIN {X 0,Y 306.2,Z 432.189,A -85,B 0,C 180,E1 -16358.923,E2 -16358.923} C_VEL
LIN {X 0,Y 308.565,Z 440.941,A -85,B 0,C 180,E1 -16360.686,E2 -16360.686} C_VEL
LIN {X 0,Y 309.935,Z 449.861,A -85,B 0,C 180,E1 -16362.515,E2 -16362.515} C_VEL
LIN {X 0,Y 310.038,Z 454.299,A -85,B 0,C 180,E1 -16363.429,E2 -16363.429} C_VEL
LIN {X 0,Y 308.048,Z 461.447,A -85,B 0,C 180,E1 -16364.789,E2 -16364.789} C_VEL
LIN {X 0,Y 305.945,Z 468.116,A -85,B 0,C 180,E1 -16366.381,E2 -16366.381} C_VEL
LIN {X 0,Y 304.136,Z 473.435,A -85,B 0,C 180,E1 -16367.996,E2 -16367.996} C_VEL
LIN {X 0,Y 302.21,Z 478.239,A -85,B 0,C 180,E1 -16369.955,E2 -16369.955} C_VEL
LIN {X 0,Y 300.515,Z 481.518,A -85,B 0,C 180,E1 -16371.934,E2 -16371.934} C_VEL
LIN {X 0,Y 299.584,Z 482.93,A -85,B 0,C 180,E1 -16373.264,E2 -16373.264} C_VEL
LIN {X 0,Y 298.798,Z 483.727,A -85,B 0,C 180,E1 -16374.602,E2 -16374.602} C_VEL
LIN {X 0,Y 298.147,Z 483.907,A -85,B 0,C 180,E1 -16375.945,E2 -16375.945} C_VEL
LIN {X 0,Y 297.751,Z 483.441,A -85,B 0,C 180,E1 -16377.294,E2 -16377.294} C_VEL
LIN {X 0,Y 297.448,Z 482.358,A -85,B 0,C 180,E1 -16378.646,E2 -16378.646} C_VEL
LIN {X 0,Y 297.228,Z 479.539,A -85,B 0,C 180,E1 -16380.678,E2 -16380.678} C_VEL
LIN {X 0,Y 297.232,Z 475.182,A -85,B 0,C 180,E1 -16382.711,E2 -16382.711} C_VEL
LIN {X 0,Y 297.472,Z 470.25,A -85,B 0,C 180,E1 -16384.404,E2 -16384.404} C_VEL
LIN {X 0,Y 297.823,Z 463.929,A -85,B 0,C 180,E1 -16386.096,E2 -16386.096} C_VEL
LIN {X 0,Y 298.092,Z 455.732,A -85,B 0,C 180,E1 -16387.819,E2 -16387.819} C_VEL
LIN {X 0,Y 298.478,Z 446.603,A -85,B 0,C 180,E1 -16389.316,E2 -16389.316} C_VEL
LIN {X 0,Y 299.017,Z 436.104,A -85,B 0,C 180,E1 -16390.667,E2 -16390.667} C_VEL
LIN {X 0,Y 299.156,Z 431.362,A -85,B 0,C 180,E1 -16391.176,E2 -16391.176} C_VEL
LIN {X 0,Y 297.894,Z 420.264,A -85,B 0,C 180,E1 -16392.173,E2 -16392.173} C_VEL
LIN {X 0,Y 297.273,Z 413.393,A -85,B 0,C 180,E1 -16392.675,E2 -16392.675} C_VEL
LIN {X 0,Y 297.462,Z 407.227,A -85,B 0,C 180,E1 -16396.471,E2 -16396.471} C_VEL
LIN {X 0,Y 297.827,Z 400.442,A -85,B 0,C 180,E1 -16400.73,E2 -16400.73} C_VEL
LIN {X 0,Y 298.166,Z 394.794,A -85,B 0,C 180,E1 -16404.362,E2 -16404.362} C_VEL
LIN {X 0,Y 298.667,Z 388.034,A -85,B 0,C 180,E1 -16408.788,E2 -16408.788} C_VEL
LIN {X 0,Y 298.758,Z 383.85,A -85,B 0,C 180,E1 -16411.615,E2 -16411.615} C_VEL
LIN {X 0,Y 298.611,Z 383.289,A -85,B 0,C 180,E1 -16412.082,E2 -16412.082} C_VEL
LIN {X 0,Y 298.448,Z 383.31,A -85,B 0,C 180,E1 -16416.807,E2 -16416.807} C_VEL
LIN {X 0,Y 298.39,Z 383.316,A -85,B 0,C 180,E1 -16421.088,E2 -16421.088} C_VEL
LIN {X 0,Y 298.391,Z 383.316,A -85,B 0,C 180,E1 -16425.041,E2 -16425.041} C_VEL
LIN {X 0,Y 298.391,Z 383.316,A -85,B 0,C 180,E1 -16428.912,E2 -16428.912} C_VEL
LIN {X 0,Y 298.447,Z 383.307,A -85,B 0,C 180,E1 -16433.193,E2 -16433.193} C_VEL
LIN {X 0,Y 298.398,Z 383.313,A -85,B 0,C 180,E1 -16437.2,E2 -16437.2} C_VEL
LIN {X 0,Y 298.43,Z 383.312,A -85,B 0,C 180,E1 -16440.616,E2 -16440.616} C_VEL
LIN {X 0,Y 298.481,Z 383.302,A -85,B 0,C 180,E1 -16443.476,E2 -16443.476} C_VEL
LIN {X 0,Y 298.438,Z 383.31,A -85,B 0,C 180,E1 -16446.697,E2 -16446.697} C_VEL
LIN {X 0,Y 298.543,Z 383.296,A -85,B 0,C 180,E1 -16450.757,E2 -16450.757} C_VEL
LIN {X 0,Y 298.597,Z 383.288,A -85,B 0,C 180,E1 -16454.995,E2 -16454.995} C_VEL
LIN {X 0,Y 298.595,Z 383.288,A -85,B 0,C 180,E1 -16459.147,E2 -16459.147} C_VEL
LIN {X 0,Y 298.744,Z 383.272,A -85,B 0,C 180,E1 -16461.885,E2 -16461.885} C_VEL
LIN {X 0,Y 298.66,Z 383.28,A -85,B 0,C 180,E1 -16464.599,E2 -16464.599} C_VEL
LIN {X 0,Y 298.925,Z 383.247,A -85,B 0,C 180,E1 -16468.653,E2 -16468.653} C_VEL
LIN {X 0,Y 298.927,Z 383.247,A -85,B 0,C 180,E1 -16471.347,E2 -16471.347} C_VEL
LIN {X 0,Y 298.795,Z 383.263,A -85,B 0,C 180,E1 -16476.754,E2 -16476.754} C_VEL
LIN {X 0,Y 298.683,Z 383.279,A -85,B 0,C 180,E1 -16479.48,E2 -16479.48} C_VEL
LIN {X 0,Y 298.555,Z 383.296,A -85,B 0,C 180,E1 -16483.615,E2 -16483.615} C_VEL
LIN {X 0,Y 298.552,Z 383.294,A -85,B 0,C 180,E1 -16486.408,E2 -16486.408} C_VEL
LIN {X 0,Y 298.519,Z 383.302,A -85,B 0,C 180,E1 -16489.657,E2 -16489.657} C_VEL
LIN {X 0,Y 298.46,Z 383.31,A -85,B 0,C 180,E1 -16493.597,E2 -16493.597} C_VEL
LIN {X 0,Y 298.489,Z 383.301,A -85,B 0,C 180,E1 -16496.574,E2 -16496.574} C_VEL
LIN {X 0,Y 298.418,Z 383.313,A -85,B 0,C 180,E1 -16499.641,E2 -16499.641} C_VEL
LIN {X 0,Y 298.397,Z 383.313,A -85,B 0,C 180,E1 -16502.8,E2 -16502.8} C_VEL
LIN {X 0,Y 298.467,Z 383.305,A -85,B 0,C 180,E1 -16506.812,E2 -16506.812} C_VEL
LIN {X 0,Y 298.39,Z 383.316,A -85,B 0,C 180,E1 -16511.088,E2 -16511.088} C_VEL
LIN {X 0,Y 298.4,Z 383.316,A -85,B 0,C 180,E1 -16513.103,E2 -16513.103} C_VEL
LIN {X 0,Y 298.404,Z 383.314,A -85,B 0,C 180,E1 -16516.921,E2 -16516.921} C_VEL
LIN {X 0,Y 298.4,Z 383.316,A -85,B 0,C 180,E1 -16521.007,E2 -16521.007} C_VEL
LIN {X 0,Y 298.419,Z 383.31,A -85,B 0,C 180,E1 -16523.93,E2 -16523.93} C_VEL
LIN {X 0,Y 298.397,Z 383.312,A -85,B 0,C 180,E1 -16527.983,E2 -16527.983} C_VEL
LIN {X 0,Y 298.465,Z 383.304,A -85,B 0,C 180,E1 -16531.904,E2 -16531.904} C_VEL
LIN {X 0,Y 298.488,Z 383.306,A -85,B 0,C 180,E1 -16534.924,E2 -16534.924} C_VEL
LIN {X 0,Y 298.452,Z 383.307,A -85,B 0,C 180,E1 -16539.315,E2 -16539.315} C_VEL
LIN {X 0,Y 298.54,Z 383.295,A -85,B 0,C 180,E1 -16542.179,E2 -16542.179} C_VEL
LIN {X 0,Y 298.596,Z 383.291,A -85,B 0,C 180,E1 -16544.995,E2 -16544.995} C_VEL
LIN {X 0,Y 298.598,Z 383.289,A -85,B 0,C 180,E1 -16549.147,E2 -16549.147} C_VEL
LIN {X 0,Y 298.76,Z 383.267,A -85,B 0,C 180,E1 -16551.886,E2 -16551.886} C_VEL
LIN {X 0,Y 298.662,Z 383.285,A -85,B 0,C 180,E1 -16554.599,E2 -16554.599} C_VEL
LIN {X 0,Y 298.926,Z 383.25,A -85,B 0,C 180,E1 -16558.653,E2 -16558.653} C_VEL
LIN {X 0,Y 298.928,Z 383.246,A -85,B 0,C 180,E1 -16561.347,E2 -16561.347} C_VEL
LIN {X 0,Y 298.663,Z 383.279,A -85,B 0,C 180,E1 -16565.401,E2 -16565.401} C_VEL
LIN {X 0,Y 298.776,Z 383.265,A -85,B 0,C 180,E1 -16567.059,E2 -16567.059} C_VEL
LIN {X 0,Y 298.05,Z 383.359,A -85,B 0,C 180,E1 -16568.183,E2 -16568.183} C_VEL
LIN {X 0,Y 295.116,Z 383.723,A -85,B 0,C 180,E1 -16570.011,E2 -16570.011} C_VEL
LIN {X 0,Y 292.651,Z 384.031,A -85,B 0,C 180,E1 -16571.494,E2 -16571.494} C_VEL
LIN {X 0,Y 291.591,Z 384.163,A -85,B 0,C 180,E1 -16572.645,E2 -16572.645} C_VEL
LIN {X 0,Y 291.502,Z 384.172,A -85,B 0,C 180,E1 -16573.035,E2 -16573.035} C_VEL
LIN {X 0,Y 291.557,Z 384.164,A -85,B 0,C 180,E1 -16575.376,E2 -16575.376} C_VEL
LIN {X 0,Y 291.452,Z 384.18,A -85,B 0,C 180,E1 -16579.875,E2 -16579.875} C_VEL
LIN {X 0,Y 291.402,Z 384.187,A -85,B 0,C 180,E1 -16584.205,E2 -16584.205} C_VEL
LIN {X 0,Y 291.422,Z 384.181,A -85,B 0,C 180,E1 -16587.272,E2 -16587.272} C_VEL
LIN {X 0,Y 291.335,Z 384.194,A -85,B 0,C 180,E1 -16590.437,E2 -16590.437} C_VEL
LIN {X 0,Y 291.346,Z 384.193,A -85,B 0,C 180,E1 -16593.698,E2 -16593.698} C_VEL
LIN {X 0,Y 291.395,Z 384.185,A -85,B 0,C 180,E1 -16597.259,E2 -16597.259} C_VEL
LIN {X 0,Y 291.337,Z 384.192,A -85,B 0,C 180,E1 -16600.642,E2 -16600.642} C_VEL
LIN {X 0,Y 291.315,Z 384.195,A -85,B 0,C 180,E1 -16604.397,E2 -16604.397} C_VEL
LIN {X 0,Y 291.389,Z 384.185,A -85,B 0,C 180,E1 -16608.7,E2 -16608.7} C_VEL
LIN {X 0,Y 293.203,Z 393.271,A -85,B 0,C 180,E1 -16612.775,E2 -16612.775} C_VEL
LIN {X 0,Y 295.388,Z 403.78,A -85,B 0,C 180,E1 -16617.229,E2 -16617.229} C_VEL
LIN {X 0,Y 296.128,Z 407.344,A -85,B 0,C 180,E1 -16618.692,E2 -16618.692} C_VEL
LIN {X 0,Y 296.259,Z 409.176,A -85,B 0,C 180,E1 -16619.417,E2 -16619.417} C_VEL
LIN {X 0,Y 294.373,Z 418.636,A -85,B 0,C 180,E1 -16623.024,E2 -16623.024} C_VEL
LIN {X 0,Y 292.46,Z 430.121,A -85,B 0,C 180,E1 -16627.388,E2 -16627.388} C_VEL
LIN {X 0,Y 291.407,Z 439.009,A -85,B 0,C 180,E1 -16630.77,E2 -16630.77} C_VEL
LIN {X 0,Y 291.784,Z 451.439,A -85,B 0,C 180,E1 -16631.389,E2 -16631.389} C_VEL
LIN {X 0,Y 292.533,Z 463.579,A -85,B 0,C 180,E1 -16632.253,E2 -16632.253} C_VEL
LIN {X 0,Y 293.156,Z 472.823,A -85,B 0,C 180,E1 -16633.101,E2 -16633.101} C_VEL
LIN {X 0,Y 292.444,Z 484.635,A -85,B 0,C 180,E1 -16634.471,E2 -16634.471} C_VEL
LIN {X 0,Y 291.675,Z 494.267,A -85,B 0,C 180,E1 -16635.879,E2 -16635.879} C_VEL
LIN {X 0,Y 291.151,Z 503.004,A -85,B 0,C 180,E1 -16637.453,E2 -16637.453} C_VEL
LIN {X 0,Y 290.676,Z 510.942,A -85,B 0,C 180,E1 -16639.2,E2 -16639.2} C_VEL
LIN {X 0,Y 290.397,Z 518.592,A -85,B 0,C 180,E1 -16641.3,E2 -16641.3} C_VEL
LIN {X 0,Y 290.381,Z 524.617,A -85,B 0,C 180,E1 -16643.416,E2 -16643.416} C_VEL
LIN {X 0,Y 290.394,Z 528.461,A -85,B 0,C 180,E1 -16645.141,E2 -16645.141} C_VEL
LIN {X 0,Y 290.494,Z 531.966,A -85,B 0,C 180,E1 -16647.227,E2 -16647.227} C_VEL
LIN {X 0,Y 290.448,Z 533.652,A -85,B 0,C 180,E1 -16648.614,E2 -16648.614} C_VEL
LIN {X 0,Y 290.381,Z 534.817,A -85,B 0,C 180,E1 -16650,E2 -16650} C_VEL
LIN {X 0,Y 290.362,Z 535.555,A -85,B 0,C 180,E1 -16651.387,E2 -16651.387} C_VEL
LIN {X 0,Y 290.133,Z 535.828,A -85,B 0,C 180,E1 -16652.777,E2 -16652.777} C_VEL
LIN {X 0,Y 289.829,Z 535.052,A -85,B 0,C 180,E1 -16655.566,E2 -16655.566} C_VEL
LIN {X 0,Y 289.768,Z 534.057,A -85,B 0,C 180,E1 -16656.966,E2 -16656.966} C_VEL
LIN {X 0,Y 290.046,Z 530.777,A -85,B 0,C 180,E1 -16659.766,E2 -16659.766} C_VEL
LIN {X 0,Y 290.627,Z 527.198,A -85,B 0,C 180,E1 -16661.862,E2 -16661.862} C_VEL
LIN {X 0,Y 291.804,Z 522.589,A -85,B 0,C 180,E1 -16663.937,E2 -16663.937} C_VEL
LIN {X 0,Y 293.5,Z 515.729,A -85,B 0,C 180,E1 -16666.342,E2 -16666.342} C_VEL
LIN {X 0,Y 295.557,Z 508.408,A -85,B 0,C 180,E1 -16668.365,E2 -16668.365} C_VEL
LIN {X 0,Y 298.135,Z 499.409,A -85,B 0,C 180,E1 -16670.347,E2 -16670.347} C_VEL
LIN {X 0,Y 300.976,Z 489.315,A -85,B 0,C 180,E1 -16672.119,E2 -16672.119} C_VEL
LIN {X 0,Y 302.85,Z 480.532,A -85,B 0,C 180,E1 -16673.416,E2 -16673.416} C_VEL
LIN {X 0,Y 303.865,Z 471.807,A -85,B 0,C 180,E1 -16674.602,E2 -16674.602} C_VEL
LIN {X 0,Y 303.697,Z 460.598,A -85,B 0,C 180,E1 -16676.084,E2 -16676.084} C_VEL
LIN {X 0,Y 302.48,Z 450.267,A -85,B 0,C 180,E1 -16677.437,E2 -16677.437} C_VEL
LIN {X 0,Y 300.108,Z 438.825,A -85,B 0,C 180,E1 -16678.982,E2 -16678.982} C_VEL
LIN {X 0,Y 299.253,Z 435.098,A -85,B 0,C 180,E1 -16679.476,E2 -16679.476} C_VEL
LIN {X 0,Y 301.181,Z 430.541,A -85,B 0,C 180,E1 -16681.671,E2 -16681.671} C_VEL
LIN {X 0,Y 301.832,Z 428.068,A -85,B 0,C 180,E1 -16683.045,E2 -16683.045} C_VEL
LIN {X 0,Y 301.389,Z 424.899,A -85,B 0,C 180,E1 -16685.298,E2 -16685.298} C_VEL
LIN {X 0,Y 300.837,Z 422.391,A -85,B 0,C 180,E1 -16687.412,E2 -16687.412} C_VEL
LIN {X 0,Y 300.145,Z 419.017,A -85,B 0,C 180,E1 -16690.968,E2 -16690.968} C_VEL
LIN {X 0,Y 299.732,Z 417.345,A -85,B 0,C 180,E1 -16693.375,E2 -16693.375} C_VEL
LIN {X 0,Y 299.235,Z 415.835,A -85,B 0,C 180,E1 -16696.726,E2 -16696.726} C_VEL
LIN {X 0,Y 298.784,Z 415.179,A -85,B 0,C 180,E1 -16700.573,E2 -16700.573} C_VEL
LIN {X 0,Y 298.528,Z 415.462,A -85,B 0,C 180,E1 -16703.945,E2 -16703.945} C_VEL
LIN {X 0,Y 298.109,Z 416.528,A -85,B 0,C 180,E1 -16707.164,E2 -16707.164} C_VEL
LIN {X 0,Y 297.788,Z 417.298,A -85,B 0,C 180,E1 -16708.72,E2 -16708.72} C_VEL
LIN {X 0,Y 296.834,Z 419.297,A -85,B 0,C 180,E1 -16711.736,E2 -16711.736} C_VEL
LIN {X 0,Y 295.692,Z 422.241,A -85,B 0,C 180,E1 -16715.187,E2 -16715.187} C_VEL
LIN {X 0,Y 299.671,Z 432.541,A -85,B 0,C 180,E1 -16717.598,E2 -16717.598} C_VEL
LIN {X 0,Y 301.982,Z 440.145,A -85,B 0,C 180,E1 -16719.299,E2 -16719.299} C_VEL
LIN {X 0,Y 303.689,Z 449.824,A -85,B 0,C 180,E1 -16721.416,E2 -16721.416} C_VEL
LIN {X 0,Y 303.934,Z 455.741,A -85,B 0,C 180,E1 -16722.735,E2 -16722.735} C_VEL
LIN {X 0,Y 301.541,Z 464.113,A -85,B 0,C 180,E1 -16724.453,E2 -16724.453} C_VEL
